gfCNCPoint3[8474] = {X 379.6357, Y 98.2550, Z -3.8333, A 0.000, B 0.000, C 0.000 }
gfCNCPoint3[8475] = {X 377.3857, Y 99.2021, Z -3.8333, A 0.000, B 0.000, C 0.000 }
gfCNCPoint3[8476] = {X 375.0734, Y 99.9850, Z -3.8333, A 0.000, B 0.000, C 0.000 }
gfCNCPoint3[8477] = {X 372.7108, Y 100.5996, Z -3.8333, A 0.000, B 0.000, C 0.000 }
gfCNCPoint3[8478] = {X 368.9146, Y 101.3340, Z -3.8333, A 0.000, B 0.000, C 0.000 }
gfCNCPoint3[8479] = {X 365.0874, Y 101.8851, Z -3.8333, A 0.000, B 0.000, C 0.000 }
gfCNCPoint3[8480] = {X 361.2381, Y 102.2515, Z -3.8333, A 0.000, B 0.000, C 0.000 }
gfCNCPoint3[8481] = {X 357.2381, Y 102.4918, Z -3.8333, A 0.000, B 0.000, C 0.000 }
gfCNCPoint3[8482] = {X 353.2338, Y 102.6450, Z -3.8333, A 0.000, B 0.000, C 0.000 }
gfCNCPoint3[8483] = {X 353.3454, Y 106.7235, Z -3.8333, A 0.000, B 0.000, C 0.000 }
gfCNCPoint3[8484] = {X 353.3454, Y 106.7235, Z -0.8333, A 0.000, B 0.000, C 0.000 }
gfCNCPoint3[8485] = {X 353.3454, Y 106.7235, Z 11.0000, A 0.000, B 0.000, C 0.000 }
gfCNCPoint3[8486] = {X 411.5989, Y 79.5929, Z 11.0000, A 0.000, B 0.000, C 0.000 }
gfCNCPoint3[8487] = {X 411.5989, Y 79.5929, Z -0.8333, A 0.000, B 0.000, C 0.000 }
gfCNCPoint3[8488] = {X 411.5989, Y 79.5929, Z -3.8333, A 0.000, B 0.000, C 0.000 }
gfCNCPoint3[8489] = {X 413.7992, Y 83.0287, Z -3.8333, A 0.000, B 0.000, C 0.000 }
gfCNCPoint3[8490] = {X 428.0548, Y 73.8995, Z -3.8333, A 0.000, B 0.000, C 0.000 }
gfCNCPoint3[8491] = {X 403.7555, Y 64.3655, Z -3.8333, A 0.000, B 0.000, C 0.000 }
gfCNCPoint3[8492] = {X 402.0596, Y 63.8040, Z -3.8333, A 0.000, B 0.000, C 0.000 }
gfCNCPoint3[8493] = {X 400.3124, Y 63.4320, Z -3.8333, A 0.000, B 0.000, C 0.000 }
gfCNCPoint3[8494] = {X 398.5348, Y 63.2540, Z -3.8333, A 0.000, B 0.000, C 0.000 }
gfCNCPoint3[8495] = {X 397.5823, Y 63.1425, Z -3.8333, A 0.000, B 0.000, C 0.000 }
gfCNCPoint3[8496] = {X 396.6778, Y 62.8236, Z -3.8333, A 0.000, B 0.000, C 0.000 }
gfCNCPoint3[8497] = {X 395.8660, Y 62.3130, Z -3.8333, A 0.000, B 0.000, C 0.000 }
gfCNCPoint3[8498] = {X 395.1868, Y 61.6358, Z -3.8333, A 0.000, B 0.000, C 0.000 }
gfCNCPoint3[8499] = {X 394.6738, Y 60.8255, Z -3.8333, A 0.000, B 0.000, C 0.000 }
gfCNCPoint3[8500] = {X 394.3522, Y 59.9220, Z -3.8333, A 0.000, B 0.000, C 0.000 }
gfCNCPoint3[8501] = {X 394.2379, Y 58.9697, Z -3.8333, A 0.000, B 0.000, C 0.000 }
gfCNCPoint3[8502] = {X 394.2377, Y 58.0000, Z -3.8333, A 0.000, B 0.000, C 0.000 }
gfCNCPoint3[8503] = {X 394.3460, Y 57.0387, Z -3.8333, A 0.000, B 0.000, C 0.000 }
gfCNCPoint3[8504] = {X 394.6655, Y 56.1256, Z -3.8333, A 0.000, B 0.000, C 0.000 }
gfCNCPoint3[8505] = {X 395.1802, Y 55.3065, Z -3.8333, A 0.000, B 0.000, C 0.000 }
gfCNCPoint3[8506] = {X 395.8642, Y 54.6225, Z -3.8333, A 0.000, B 0.000, C 0.000 }
gfCNCPoint3[8507] = {X 396.6833, Y 54.1078, Z -3.8333, A 0.000, B 0.000, C 0.000 }
gfCNCPoint3[8508] = {X 397.5964, Y 53.7883, Z -3.8333, A 0.000, B 0.000, C 0.000 }
gfCNCPoint3[8509] = {X 398.5577, Y 53.6800, Z -3.8333, A 0.000, B 0.000, C 0.000 }
gfCNCPoint3[8510] = {X 419.4886, Y 53.6800, Z -3.8333, A 0.000, B 0.000, C 0.000 }
gfCNCPoint3[8511] = {X 420.4499, Y 53.7883, Z -3.8333, A 0.000, B 0.000, C 0.000 }
gfCNCPoint3[8512] = {X 421.3630, Y 54.1078, Z -3.8333, A 0.000, B 0.000, C 0.000 }
gfCNCPoint3[8513] = {X 422.1821, Y 54.6225, Z -3.8333, A 0.000, B 0.000, C 0.000 }
gfCNCPoint3[8514] = {X 422.8661, Y 55.3065, Z -3.8333, A 0.000, B 0.000, C 0.000 }
gfCNCPoint3[8515] = {X 423.3808, Y 56.1256, Z -3.8333, A 0.000, B 0.000, C 0.000 }
gfCNCPoint3[8516] = {X 423.7003, Y 57.0387, Z -3.8333, A 0.000, B 0.000, C 0.000 }
gfCNCPoint3[8517] = {X 423.8086, Y 58.0000, Z -3.8333, A 0.000, B 0.000, C 0.000 }
gfCNCPoint3[8518] = {X 423.8086, Y 58.2323, Z -3.8333, A 0.000, B 0.000, C 0.000 }
gfCNCPoint3[8519] = {X 429.6116, Y 60.4937, Z -3.8333, A 0.000, B 0.000, C 0.000 }
gfCNCPoint3[8520] = {X 457.8588, Y 71.7009, Z -3.8333, A 0.000, B 0.000, C 0.000 }
gfCNCPoint3[8521] = {X 457.8609, Y 63.2124, Z -3.8333, A 0.000, B 0.000, C 0.000 }
gfCNCPoint3[8522] = {X 457.0092, Y 63.0033, Z -3.8333, A 0.000, B 0.000, C 0.000 }
gfCNCPoint3[8523] = {X 456.2172, Y 62.6265, Z -3.8333, A 0.000, B 0.000, C 0.000 }
gfCNCPoint3[8524] = {X 455.5177, Y 62.0976, Z -3.8333, A 0.000, B 0.000, C 0.000 }
gfCNCPoint3[8525] = {X 454.9395, Y 61.4383, Z -3.8333, A 0.000, B 0.000, C 0.000 }
gfCNCPoint3[8526] = {X 454.5063, Y 60.6757, Z -3.8333, A 0.000, B 0.000, C 0.000 }
gfCNCPoint3[8527] = {X 454.2360, Y 59.8414, Z -3.8333, A 0.000, B 0.000, C 0.000 }
gfCNCPoint3[8528] = {X 454.1398, Y 58.9697, Z -3.8333, A 0.000, B 0.000, C 0.000 }
gfCNCPoint3[8529] = {X 454.1396, Y 58.0000, Z -3.8333, A 0.000, B 0.000, C 0.000 }
gfCNCPoint3[8530] = {X 454.2479, Y 57.0387, Z -3.8333, A 0.000, B 0.000, C 0.000 }
gfCNCPoint3[8531] = {X 454.5674, Y 56.1256, Z -3.8333, A 0.000, B 0.000, C 0.000 }
gfCNCPoint3[8532] = {X 455.0821, Y 55.3065, Z -3.8333, A 0.000, B 0.000, C 0.000 }
gfCNCPoint3[8533] = {X 455.7661, Y 54.6225, Z -3.8333, A 0.000, B 0.000, C 0.000 }
gfCNCPoint3[8534] = {X 456.5852, Y 54.1078, Z -3.8333, A 0.000, B 0.000, C 0.000 }
gfCNCPoint3[8535] = {X 457.4983, Y 53.7883, Z -3.8333, A 0.000, B 0.000, C 0.000 }
gfCNCPoint3[8536] = {X 458.4596, Y 53.6800, Z -3.8333, A 0.000, B 0.000, C 0.000 }
gfCNCPoint3[8537] = {X 475.0000, Y 53.6800, Z -3.8333, A 0.000, B 0.000, C 0.000 }
gfCNCPoint3[8538] = {X 475.9613, Y 53.7883, Z -3.8333, A 0.000, B 0.000, C 0.000 }
gfCNCPoint3[8539] = {X 476.8744, Y 54.1078, Z -3.8333, A 0.000, B 0.000, C 0.000 }
gfCNCPoint3[8540] = {X 477.6935, Y 54.6225, Z -3.8333, A 0.000, B 0.000, C 0.000 }
gfCNCPoint3[8541] = {X 478.3775, Y 55.3065, Z -3.8333, A 0.000, B 0.000, C 0.000 }
gfCNCPoint3[8542] = {X 478.8922, Y 56.1256, Z -3.8333, A 0.000, B 0.000, C 0.000 }
gfCNCPoint3[8543] = {X 479.2117, Y 57.0387, Z -3.8333, A 0.000, B 0.000, C 0.000 }
gfCNCPoint3[8544] = {X 479.3200, Y 58.0000, Z -3.8333, A 0.000, B 0.000, C 0.000 }
gfCNCPoint3[8545] = {X 479.3200, Y 58.9342, Z -3.8333, A 0.000, B 0.000, C 0.000 }
gfCNCPoint3[8546] = {X 479.2300, Y 59.8115, Z -3.8333, A 0.000, B 0.000, C 0.000 }
gfCNCPoint3[8547] = {X 478.9637, Y 60.6522, Z -3.8333, A 0.000, B 0.000, C 0.000 }
gfCNCPoint3[8548] = {X 478.5322, Y 61.4212, Z -3.8333, A 0.000, B 0.000, C 0.000 }
gfCNCPoint3[8549] = {X 477.9535, Y 62.0867, Z -3.8333, A 0.000, B 0.000, C 0.000 }
gfCNCPoint3[8550] = {X 477.2518, Y 62.6208, Z -3.8333, A 0.000, B 0.000, C 0.000 }
gfCNCPoint3[8551] = {X 476.4562, Y 63.0012, Z -3.8333, A 0.000, B 0.000, C 0.000 }
gfCNCPoint3[8552] = {X 475.6000, Y 63.2122, Z -3.8333, A 0.000, B 0.000, C 0.000 }
gfCNCPoint3[8553] = {X 475.6004, Y 92.7684, Z -3.8333, A 0.000, B 0.000, C 0.000 }
gfCNCPoint3[8554] = {X 475.9967, Y 92.8675, Z -3.8333, A 0.000, B 0.000, C 0.000 }
gfCNCPoint3[8555] = {X 476.3874, Y 92.9869, Z -3.8333, A 0.000, B 0.000, C 0.000 }
gfCNCPoint3[8556] = {X 477.1991, Y 93.3557, Z -3.8333, A 0.000, B 0.000, C 0.000 }
gfCNCPoint3[8557] = {X 477.9172, Y 93.8843, Z -3.8333, A 0.000, B 0.000, C 0.000 }
gfCNCPoint3[8558] = {X 478.5105, Y 94.5498, Z -3.8333, A 0.000, B 0.000, C 0.000 }
gfCNCPoint3[8559] = {X 478.9537, Y 95.3235, Z -3.8333, A 0.000, B 0.000, C 0.000 }
gfCNCPoint3[8560] = {X 479.2274, Y 96.1721, Z -3.8333, A 0.000, B 0.000, C 0.000 }
gfCNCPoint3[8561] = {X 479.3200, Y 97.0589, Z -3.8333, A 0.000, B 0.000, C 0.000 }
gfCNCPoint3[8562] = {X 479.3200, Y 98.0000, Z -3.8333, A 0.000, B 0.000, C 0.000 }
gfCNCPoint3[8563] = {X 479.2117, Y 98.9613, Z -3.8333, A 0.000, B 0.000, C 0.000 }
gfCNCPoint3[8564] = {X 478.8922, Y 99.8744, Z -3.8333, A 0.000, B 0.000, C 0.000 }
gfCNCPoint3[8565] = {X 478.3775, Y 100.6935, Z -3.8333, A 0.000, B 0.000, C 0.000 }
gfCNCPoint3[8566] = {X 477.6935, Y 101.3775, Z -3.8333, A 0.000, B 0.000, C 0.000 }
gfCNCPoint3[8567] = {X 476.8744, Y 101.8922, Z -3.8333, A 0.000, B 0.000, C 0.000 }
gfCNCPoint3[8568] = {X 475.9613, Y 102.2117, Z -3.8333, A 0.000, B 0.000, C 0.000 }
gfCNCPoint3[8569] = {X 475.0000, Y 102.3200, Z -3.8333, A 0.000, B 0.000, C 0.000 }
gfCNCPoint3[8570] = {X 458.4596, Y 102.3200, Z -3.8333, A 0.000, B 0.000, C 0.000 }
gfCNCPoint3[8571] = {X 457.4983, Y 102.2117, Z -3.8333, A 0.000, B 0.000, C 0.000 }
gfCNCPoint3[8572] = {X 456.5852, Y 101.8922, Z -3.8333, A 0.000, B 0.000, C 0.000 }
gfCNCPoint3[8573] = {X 455.7661, Y 101.3775, Z -3.8333, A 0.000, B 0.000, C 0.000 }
gfCNCPoint3[8574] = {X 455.0821, Y 100.6935, Z -3.8333, A 0.000, B 0.000, C 0.000 }
gfCNCPoint3[8575] = {X 454.5674, Y 99.8744, Z -3.8333, A 0.000, B 0.000, C 0.000 }
gfCNCPoint3[8576] = {X 454.2479, Y 98.9613, Z -3.8333, A 0.000, B 0.000, C 0.000 }
gfCNCPoint3[8577] = {X 454.1396, Y 98.0000, Z -3.8333, A 0.000, B 0.000, C 0.000 }
gfCNCPoint3[8578] = {X 454.1396, Y 97.0659, Z -3.8333, A 0.000, B 0.000, C 0.000 }
gfCNCPoint3[8579] = {X 454.2295, Y 96.1891, Z -3.8333, A 0.000, B 0.000, C 0.000 }
gfCNCPoint3[8580] = {X 454.4955, Y 95.3488, Z -3.8333, A 0.000, B 0.000, C 0.000 }
gfCNCPoint3[8581] = {X 454.9265, Y 94.5800, Z -3.8333, A 0.000, B 0.000, C 0.000 }
gfCNCPoint3[8582] = {X 455.5046, Y 93.9147, Z -3.8333, A 0.000, B 0.000, C 0.000 }
gfCNCPoint3[8583] = {X 456.2057, Y 93.3805, Z -3.8333, A 0.000, B 0.000, C 0.000 }
gfCNCPoint3[8584] = {X 457.0006, Y 92.9998, Z -3.8333, A 0.000, B 0.000, C 0.000 }
gfCNCPoint3[8585] = {X 457.8563, Y 92.7883, Z -3.8333, A 0.000, B 0.000, C 0.000 }
gfCNCPoint3[8586] = {X 457.8563, Y 85.5950, Z -3.8333, A 0.000, B 0.000, C 0.000 }
gfCNCPoint3[8587] = {X 444.8588, Y 80.4999, Z -3.8333, A 0.000, B 0.000, C 0.000 }
gfCNCPoint3[8588] = {X 420.0232, Y 96.5882, Z -3.8333, A 0.000, B 0.000, C 0.000 }
gfCNCPoint3[8589] = {X 420.0267, Y 97.0647, Z -3.8333, A 0.000, B 0.000, C 0.000 }
gfCNCPoint3[8590] = {X 420.0267, Y 98.0000, Z -3.8333, A 0.000, B 0.000, C 0.000 }
gfCNCPoint3[8591] = {X 419.9184, Y 98.9613, Z -3.8333, A 0.000, B 0.000, C 0.000 }
gfCNCPoint3[8592] = {X 419.5989, Y 99.8744, Z -3.8333, A 0.000, B 0.000, C 0.000 }
gfCNCPoint3[8593] = {X 419.0842, Y 100.6935, Z -3.8333, A 0.000, B 0.000, C 0.000 }
gfCNCPoint3[8594] = {X 418.4002, Y 101.3775, Z -3.8333, A 0.000, B 0.000, C 0.000 }
gfCNCPoint3[8595] = {X 417.5811, Y 101.8922, Z -3.8333, A 0.000, B 0.000, C 0.000 }
gfCNCPoint3[8596] = {X 416.6680, Y 102.2117, Z -3.8333, A 0.000, B 0.000, C 0.000 }
gfCNCPoint3[8597] = {X 415.7067, Y 102.3200, Z -3.8333, A 0.000, B 0.000, C 0.000 }
gfCNCPoint3[8598] = {X 396.4059, Y 102.3200, Z -3.8333, A 0.000, B 0.000, C 0.000 }
gfCNCPoint3[8599] = {X 395.4447, Y 102.2117, Z -3.8333, A 0.000, B 0.000, C 0.000 }
gfCNCPoint3[8600] = {X 394.5316, Y 101.8922, Z -3.8333, A 0.000, B 0.000, C 0.000 }
gfCNCPoint3[8601] = {X 393.7125, Y 101.3775, Z -3.8333, A 0.000, B 0.000, C 0.000 }
gfCNCPoint3[8602] = {X 393.0284, Y 100.6935, Z -3.8333, A 0.000, B 0.000, C 0.000 }
gfCNCPoint3[8603] = {X 392.5138, Y 99.8744, Z -3.8333, A 0.000, B 0.000, C 0.000 }
gfCNCPoint3[8604] = {X 392.1943, Y 98.9613, Z -3.8333, A 0.000, B 0.000, C 0.000 }
gfCNCPoint3[8605] = {X 392.0859, Y 98.0000, Z -3.8333, A 0.000, B 0.000, C 0.000 }
gfCNCPoint3[8606] = {X 392.0859, Y 97.0659, Z -3.8333, A 0.000, B 0.000, C 0.000 }
gfCNCPoint3[8607] = {X 392.1954, Y 96.0997, Z -3.8333, A 0.000, B 0.000, C 0.000 }
gfCNCPoint3[8608] = {X 392.5182, Y 95.1825, Z -3.8333, A 0.000, B 0.000, C 0.000 }
gfCNCPoint3[8609] = {X 393.0379, Y 94.3606, Z -3.8333, A 0.000, B 0.000, C 0.000 }
gfCNCPoint3[8610] = {X 393.7283, Y 93.6759, Z -3.8333, A 0.000, B 0.000, C 0.000 }
gfCNCPoint3[8611] = {X 394.5544, Y 93.1629, Z -3.8333, A 0.000, B 0.000, C 0.000 }
gfCNCPoint3[8612] = {X 395.4742, Y 92.8476, Z -3.8333, A 0.000, B 0.000, C 0.000 }
gfCNCPoint3[8613] = {X 396.4413, Y 92.7461, Z -3.8333, A 0.000, B 0.000, C 0.000 }
gfCNCPoint3[8614] = {X 397.3691, Y 92.7028, Z -3.8333, A 0.000, B 0.000, C 0.000 }
gfCNCPoint3[8615] = {X 398.2936, Y 92.6146, Z -3.8333, A 0.000, B 0.000, C 0.000 }
gfCNCPoint3[8616] = {X 398.9444, Y 92.4569, Z -3.8333, A 0.000, B 0.000, C 0.000 }
gfCNCPoint3[8617] = {X 399.5436, Y 92.1580, Z -3.8333, A 0.000, B 0.000, C 0.000 }
gfCNCPoint3[8618] = {X 413.7992, Y 83.0287, Z -3.8333, A 0.000, B 0.000, C 0.000 }
gfCNCPoint3[8619] = {X 411.6421, Y 79.6603, Z -3.8333, A 0.000, B 0.000, C 0.000 }
gfCNCPoint3[8620] = {X 413.8424, Y 83.0961, Z -3.8333, A 0.000, B 0.000, C 0.000 }
gfCNCPoint3[8621] = {X 428.2300, Y 73.8823, Z -3.8333, A 0.000, B 0.000, C 0.000 }
gfCNCPoint3[8622] = {X 403.7847, Y 64.2910, Z -3.8333, A 0.000, B 0.000, C 0.000 }
gfCNCPoint3[8623] = {X 402.0800, Y 63.7266, Z -3.8333, A 0.000, B 0.000, C 0.000 }
gfCNCPoint3[8624] = {X 400.3236, Y 63.3528, Z -3.8333, A 0.000, B 0.000, C 0.000 }
gfCNCPoint3[8625] = {X 398.5368, Y 63.1740, Z -3.8333, A 0.000, B 0.000, C 0.000 }
gfCNCPoint3[8626] = {X 397.6017, Y 63.0649, Z -3.8333, A 0.000, B 0.000, C 0.000 }
gfCNCPoint3[8627] = {X 396.7136, Y 62.7520, Z -3.8333, A 0.000, B 0.000, C 0.000 }
gfCNCPoint3[8628] = {X 395.9165, Y 62.2509, Z -3.8333, A 0.000, B 0.000, C 0.000 }
gfCNCPoint3[8629] = {X 395.2497, Y 61.5863, Z -3.8333, A 0.000, B 0.000, C 0.000 }
gfCNCPoint3[8630] = {X 394.7459, Y 60.7909, Z -3.8333, A 0.000, B 0.000, C 0.000 }
gfCNCPoint3[8631] = {X 394.4301, Y 59.9039, Z -3.8333, A 0.000, B 0.000, C 0.000 }
gfCNCPoint3[8632] = {X 394.3179, Y 58.9691, Z -3.8333, A 0.000, B 0.000, C 0.000 }
gfCNCPoint3[8633] = {X 394.3177, Y 58.0000, Z -3.8333, A 0.000, B 0.000, C 0.000 }
gfCNCPoint3[8634] = {X 394.4240, Y 57.0565, Z -3.8333, A 0.000, B 0.000, C 0.000 }
gfCNCPoint3[8635] = {X 394.7376, Y 56.1603, Z -3.8333, A 0.000, B 0.000, C 0.000 }
gfCNCPoint3[8636] = {X 395.2428, Y 55.3564, Z -3.8333, A 0.000, B 0.000, C 0.000 }
gfCNCPoint3[8637] = {X 395.9141, Y 54.6850, Z -3.8333, A 0.000, B 0.000, C 0.000 }
gfCNCPoint3[8638] = {X 396.7181, Y 54.1799, Z -3.8333, A 0.000, B 0.000, C 0.000 }
gfCNCPoint3[8639] = {X 397.6142, Y 53.8663, Z -3.8333, A 0.000, B 0.000, C 0.000 }
gfCNCPoint3[8640] = {X 398.5577, Y 53.7600, Z -3.8333, A 0.000, B 0.000, C 0.000 }
gfCNCPoint3[8641] = {X 419.4886, Y 53.7600, Z -3.8333, A 0.000, B 0.000, C 0.000 }
gfCNCPoint3[8642] = {X 420.4321, Y 53.8663, Z -3.8333, A 0.000, B 0.000, C 0.000 }
gfCNCPoint3[8643] = {X 421.3283, Y 54.1799, Z -3.8333, A 0.000, B 0.000, C 0.000 }
gfCNCPoint3[8644] = {X 422.1322, Y 54.6850, Z -3.8333, A 0.000, B 0.000, C 0.000 }
gfCNCPoint3[8645] = {X 422.8036, Y 55.3564, Z -3.8333, A 0.000, B 0.000, C 0.000 }
gfCNCPoint3[8646] = {X 423.3087, Y 56.1603, Z -3.8333, A 0.000, B 0.000, C 0.000 }
gfCNCPoint3[8647] = {X 423.6223, Y 57.0565, Z -3.8333, A 0.000, B 0.000, C 0.000 }
gfCNCPoint3[8648] = {X 423.7286, Y 58.0000, Z -3.8333, A 0.000, B 0.000, C 0.000 }
gfCNCPoint3[8649] = {X 423.7286, Y 58.2870, Z -3.8333, A 0.000, B 0.000, C 0.000 }
gfCNCPoint3[8650] = {X 429.5823, Y 60.5682, Z -3.8333, A 0.000, B 0.000, C 0.000 }
gfCNCPoint3[8651] = {X 457.9388, Y 71.8187, Z -3.8333, A 0.000, B 0.000, C 0.000 }
gfCNCPoint3[8652] = {X 457.9409, Y 63.1422, Z -3.8333, A 0.000, B 0.000, C 0.000 }
gfCNCPoint3[8653] = {X 457.0923, Y 62.9476, Z -3.8333, A 0.000, B 0.000, C 0.000 }
gfCNCPoint3[8654] = {X 456.3014, Y 62.5837, Z -3.8333, A 0.000, B 0.000, C 0.000 }
gfCNCPoint3[8655] = {X 455.6014, Y 62.0659, Z -3.8333, A 0.000, B 0.000, C 0.000 }
gfCNCPoint3[8656] = {X 455.0220, Y 61.4161, Z -3.8333, A 0.000, B 0.000, C 0.000 }
gfCNCPoint3[8657] = {X 454.5875, Y 60.6616, Z -3.8333, A 0.000, B 0.000, C 0.000 }
gfCNCPoint3[8658] = {X 454.3163, Y 59.8343, Z -3.8333, A 0.000, B 0.000, C 0.000 }
gfCNCPoint3[8659] = {X 454.2197, Y 58.9691, Z -3.8333, A 0.000, B 0.000, C 0.000 }
gfCNCPoint3[8660] = {X 454.2196, Y 58.0000, Z -3.8333, A 0.000, B 0.000, C 0.000 }
gfCNCPoint3[8661] = {X 454.3259, Y 57.0565, Z -3.8333, A 0.000, B 0.000, C 0.000 }
gfCNCPoint3[8662] = {X 454.6395, Y 56.1603, Z -3.8333, A 0.000, B 0.000, C 0.000 }
gfCNCPoint3[8663] = {X 455.1446, Y 55.3564, Z -3.8333, A 0.000, B 0.000, C 0.000 }
gfCNCPoint3[8664] = {X 455.8160, Y 54.6850, Z -3.8333, A 0.000, B 0.000, C 0.000 }
gfCNCPoint3[8665] = {X 456.6199, Y 54.1799, Z -3.8333, A 0.000, B 0.000, C 0.000 }
gfCNCPoint3[8666] = {X 457.5161, Y 53.8663, Z -3.8333, A 0.000, B 0.000, C 0.000 }
gfCNCPoint3[8667] = {X 458.4596, Y 53.7600, Z -3.8333, A 0.000, B 0.000, C 0.000 }
gfCNCPoint3[8668] = {X 475.0000, Y 53.7600, Z -3.8333, A 0.000, B 0.000, C 0.000 }
gfCNCPoint3[8669] = {X 475.9435, Y 53.8663, Z -3.8333, A 0.000, B 0.000, C 0.000 }
gfCNCPoint3[8670] = {X 476.8397, Y 54.1799, Z -3.8333, A 0.000, B 0.000, C 0.000 }
gfCNCPoint3[8671] = {X 477.6436, Y 54.6850, Z -3.8333, A 0.000, B 0.000, C 0.000 }
gfCNCPoint3[8672] = {X 478.3150, Y 55.3564, Z -3.8333, A 0.000, B 0.000, C 0.000 }
gfCNCPoint3[8673] = {X 478.8201, Y 56.1603, Z -3.8333, A 0.000, B 0.000, C 0.000 }
gfCNCPoint3[8674] = {X 479.1337, Y 57.0565, Z -3.8333, A 0.000, B 0.000, C 0.000 }
gfCNCPoint3[8675] = {X 479.2400, Y 58.0000, Z -3.8333, A 0.000, B 0.000, C 0.000 }
gfCNCPoint3[8676] = {X 479.2400, Y 58.9342, Z -3.8333, A 0.000, B 0.000, C 0.000 }
gfCNCPoint3[8677] = {X 479.1496, Y 59.8049, Z -3.8333, A 0.000, B 0.000, C 0.000 }
gfCNCPoint3[8678] = {X 478.8823, Y 60.6385, Z -3.8333, A 0.000, B 0.000, C 0.000 }
gfCNCPoint3[8679] = {X 478.4495, Y 61.3995, Z -3.8333, A 0.000, B 0.000, C 0.000 }
gfCNCPoint3[8680] = {X 477.8697, Y 62.0553, Z -3.8333, A 0.000, B 0.000, C 0.000 }
gfCNCPoint3[8681] = {X 477.1676, Y 62.5781, Z -3.8333, A 0.000, B 0.000, C 0.000 }
gfCNCPoint3[8682] = {X 476.3730, Y 62.9456, Z -3.8333, A 0.000, B 0.000, C 0.000 }
gfCNCPoint3[8683] = {X 475.5200, Y 63.1421, Z -3.8333, A 0.000, B 0.000, C 0.000 }
gfCNCPoint3[8684] = {X 475.5204, Y 92.8328, Z -3.8333, A 0.000, B 0.000, C 0.000 }
gfCNCPoint3[8685] = {X 475.9444, Y 92.9360, Z -3.8333, A 0.000, B 0.000, C 0.000 }
gfCNCPoint3[8686] = {X 476.3620, Y 93.0628, Z -3.8333, A 0.000, B 0.000, C 0.000 }
gfCNCPoint3[8687] = {X 477.1586, Y 93.4247, Z -3.8333, A 0.000, B 0.000, C 0.000 }
gfCNCPoint3[8688] = {X 477.8633, Y 93.9435, Z -3.8333, A 0.000, B 0.000, C 0.000 }
gfCNCPoint3[8689] = {X 478.4456, Y 94.5966, Z -3.8333, A 0.000, B 0.000, C 0.000 }
gfCNCPoint3[8690] = {X 478.8805, Y 95.3559, Z -3.8333, A 0.000, B 0.000, C 0.000 }
gfCNCPoint3[8691] = {X 479.1491, Y 96.1886, Z -3.8333, A 0.000, B 0.000, C 0.000 }
gfCNCPoint3[8692] = {X 479.2400, Y 97.0589, Z -3.8333, A 0.000, B 0.000, C 0.000 }
gfCNCPoint3[8693] = {X 479.2400, Y 98.0000, Z -3.8333, A 0.000, B 0.000, C 0.000 }
gfCNCPoint3[8694] = {X 479.1337, Y 98.9435, Z -3.8333, A 0.000, B 0.000, C 0.000 }
gfCNCPoint3[8695] = {X 478.8201, Y 99.8397, Z -3.8333, A 0.000, B 0.000, C 0.000 }
gfCNCPoint3[8696] = {X 478.3150, Y 100.6436, Z -3.8333, A 0.000, B 0.000, C 0.000 }
gfCNCPoint3[8697] = {X 477.6436, Y 101.3150, Z -3.8333, A 0.000, B 0.000, C 0.000 }
gfCNCPoint3[8698] = {X 476.8397, Y 101.8201, Z -3.8333, A 0.000, B 0.000, C 0.000 }
gfCNCPoint3[8699] = {X 475.9435, Y 102.1337, Z -3.8333, A 0.000, B 0.000, C 0.000 }
gfCNCPoint3[8700] = {X 475.0000, Y 102.2400, Z -3.8333, A 0.000, B 0.000, C 0.000 }
gfCNCPoint3[8701] = {X 458.4596, Y 102.2400, Z -3.8333, A 0.000, B 0.000, C 0.000 }
gfCNCPoint3[8702] = {X 457.5161, Y 102.1337, Z -3.8333, A 0.000, B 0.000, C 0.000 }
gfCNCPoint3[8703] = {X 456.6199, Y 101.8201, Z -3.8333, A 0.000, B 0.000, C 0.000 }
gfCNCPoint3[8704] = {X 455.8160, Y 101.3150, Z -3.8333, A 0.000, B 0.000, C 0.000 }
gfCNCPoint3[8705] = {X 455.1446, Y 100.6436, Z -3.8333, A 0.000, B 0.000, C 0.000 }
gfCNCPoint3[8706] = {X 454.6395, Y 99.8397, Z -3.8333, A 0.000, B 0.000, C 0.000 }
gfCNCPoint3[8707] = {X 454.3259, Y 98.9435, Z -3.8333, A 0.000, B 0.000, C 0.000 }
gfCNCPoint3[8708] = {X 454.2196, Y 98.0000, Z -3.8333, A 0.000, B 0.000, C 0.000 }
gfCNCPoint3[8709] = {X 454.2196, Y 97.0659, Z -3.8333, A 0.000, B 0.000, C 0.000 }
gfCNCPoint3[8710] = {X 454.3099, Y 96.1957, Z -3.8333, A 0.000, B 0.000, C 0.000 }
gfCNCPoint3[8711] = {X 454.5769, Y 95.3624, Z -3.8333, A 0.000, B 0.000, C 0.000 }
gfCNCPoint3[8712] = {X 455.0092, Y 94.6018, Z -3.8333, A 0.000, B 0.000, C 0.000 }
gfCNCPoint3[8713] = {X 455.5884, Y 93.9460, Z -3.8333, A 0.000, B 0.000, C 0.000 }
gfCNCPoint3[8714] = {X 456.2899, Y 93.4231, Z -3.8333, A 0.000, B 0.000, C 0.000 }
gfCNCPoint3[8715] = {X 457.0838, Y 93.0553, Z -3.8333, A 0.000, B 0.000, C 0.000 }
gfCNCPoint3[8716] = {X 457.9363, Y 92.8584, Z -3.8333, A 0.000, B 0.000, C 0.000 }
gfCNCPoint3[8717] = {X 457.9363, Y 85.5404, Z -3.8333, A 0.000, B 0.000, C 0.000 }
gfCNCPoint3[8718] = {X 444.8498, Y 80.4105, Z -3.8333, A 0.000, B 0.000, C 0.000 }
gfCNCPoint3[8719] = {X 419.9429, Y 96.5449, Z -3.8333, A 0.000, B 0.000, C 0.000 }
gfCNCPoint3[8720] = {X 419.9467, Y 97.0650, Z -3.8333, A 0.000, B 0.000, C 0.000 }
gfCNCPoint3[8721] = {X 419.9467, Y 98.0000, Z -3.8333, A 0.000, B 0.000, C 0.000 }
gfCNCPoint3[8722] = {X 419.8404, Y 98.9435, Z -3.8333, A 0.000, B 0.000, C 0.000 }
gfCNCPoint3[8723] = {X 419.5268, Y 99.8397, Z -3.8333, A 0.000, B 0.000, C 0.000 }
gfCNCPoint3[8724] = {X 419.0217, Y 100.6436, Z -3.8333, A 0.000, B 0.000, C 0.000 }
gfCNCPoint3[8725] = {X 418.3503, Y 101.3150, Z -3.8333, A 0.000, B 0.000, C 0.000 }
gfCNCPoint3[8726] = {X 417.5464, Y 101.8201, Z -3.8333, A 0.000, B 0.000, C 0.000 }
gfCNCPoint3[8727] = {X 416.6502, Y 102.1337, Z -3.8333, A 0.000, B 0.000, C 0.000 }
gfCNCPoint3[8728] = {X 415.7067, Y 102.2400, Z -3.8333, A 0.000, B 0.000, C 0.000 }
gfCNCPoint3[8729] = {X 396.4059, Y 102.2400, Z -3.8333, A 0.000, B 0.000, C 0.000 }
gfCNCPoint3[8730] = {X 395.4625, Y 102.1337, Z -3.8333, A 0.000, B 0.000, C 0.000 }
gfCNCPoint3[8731] = {X 394.5663, Y 101.8201, Z -3.8333, A 0.000, B 0.000, C 0.000 }
gfCNCPoint3[8732] = {X 393.7624, Y 101.3150, Z -3.8333, A 0.000, B 0.000, C 0.000 }
gfCNCPoint3[8733] = {X 393.0910, Y 100.6436, Z -3.8333, A 0.000, B 0.000, C 0.000 }
gfCNCPoint3[8734] = {X 392.5858, Y 99.8397, Z -3.8333, A 0.000, B 0.000, C 0.000 }
gfCNCPoint3[8735] = {X 392.2723, Y 98.9435, Z -3.8333, A 0.000, B 0.000, C 0.000 }
gfCNCPoint3[8736] = {X 392.1659, Y 98.0000, Z -3.8333, A 0.000, B 0.000, C 0.000 }
gfCNCPoint3[8737] = {X 392.1659, Y 97.0659, Z -3.8333, A 0.000, B 0.000, C 0.000 }
gfCNCPoint3[8738] = {X 392.2734, Y 96.1174, Z -3.8333, A 0.000, B 0.000, C 0.000 }
gfCNCPoint3[8739] = {X 392.5903, Y 95.2170, Z -3.8333, A 0.000, B 0.000, C 0.000 }
gfCNCPoint3[8740] = {X 393.1006, Y 94.4103, Z -3.8333, A 0.000, B 0.000, C 0.000 }
gfCNCPoint3[8741] = {X 393.7784, Y 93.7382, Z -3.8333, A 0.000, B 0.000, C 0.000 }
gfCNCPoint3[8742] = {X 394.5894, Y 93.2348, Z -3.8333, A 0.000, B 0.000, C 0.000 }
gfCNCPoint3[8743] = {X 395.4925, Y 92.9255, Z -3.8333, A 0.000, B 0.000, C 0.000 }
gfCNCPoint3[8744] = {X 396.4419, Y 92.8261, Z -3.8333, A 0.000, B 0.000, C 0.000 }
gfCNCPoint3[8745] = {X 397.3742, Y 92.7827, Z -3.8333, A 0.000, B 0.000, C 0.000 }
gfCNCPoint3[8746] = {X 398.3034, Y 92.6940, Z -3.8333, A 0.000, B 0.000, C 0.000 }
gfCNCPoint3[8747] = {X 398.9717, Y 92.5321, Z -3.8333, A 0.000, B 0.000, C 0.000 }
gfCNCPoint3[8748] = {X 399.5871, Y 92.2251, Z -3.8333, A 0.000, B 0.000, C 0.000 }
gfCNCPoint3[8749] = {X 413.8424, Y 83.0961, Z -3.8333, A 0.000, B 0.000, C 0.000 }
gfCNCPoint3[8750] = {X 411.6852, Y 79.7276, Z -3.8333, A 0.000, B 0.000, C 0.000 }
gfCNCPoint3[8751] = {X 413.8855, Y 83.1635, Z -3.8333, A 0.000, B 0.000, C 0.000 }
gfCNCPoint3[8752] = {X 428.4052, Y 73.8651, Z -3.8333, A 0.000, B 0.000, C 0.000 }
gfCNCPoint3[8753] = {X 403.8140, Y 64.2166, Z -3.8333, A 0.000, B 0.000, C 0.000 }
gfCNCPoint3[8754] = {X 402.1004, Y 63.6493, Z -3.8333, A 0.000, B 0.000, C 0.000 }
gfCNCPoint3[8755] = {X 400.3349, Y 63.2736, Z -3.8333, A 0.000, B 0.000, C 0.000 }
gfCNCPoint3[8756] = {X 398.5388, Y 63.0940, Z -3.8333, A 0.000, B 0.000, C 0.000 }
gfCNCPoint3[8757] = {X 397.6210, Y 62.9872, Z -3.8333, A 0.000, B 0.000, C 0.000 }
gfCNCPoint3[8758] = {X 396.7494, Y 62.6805, Z -3.8333, A 0.000, B 0.000, C 0.000 }
gfCNCPoint3[8759] = {X 395.9671, Y 62.1889, Z -3.8333, A 0.000, B 0.000, C 0.000 }
gfCNCPoint3[8760] = {X 395.3125, Y 61.5368, Z -3.8333, A 0.000, B 0.000, C 0.000 }
gfCNCPoint3[8761] = {X 394.8180, Y 60.7562, Z -3.8333, A 0.000, B 0.000, C 0.000 }
gfCNCPoint3[8762] = {X 394.5081, Y 59.8858, Z -3.8333, A 0.000, B 0.000, C 0.000 }
gfCNCPoint3[8763] = {X 394.3979, Y 58.9684, Z -3.8333, A 0.000, B 0.000, C 0.000 }
gfCNCPoint3[8764] = {X 394.3977, Y 58.0000, Z -3.8333, A 0.000, B 0.000, C 0.000 }
gfCNCPoint3[8765] = {X 394.5020, Y 57.0743, Z -3.8333, A 0.000, B 0.000, C 0.000 }
gfCNCPoint3[8766] = {X 394.8097, Y 56.1950, Z -3.8333, A 0.000, B 0.000, C 0.000 }
gfCNCPoint3[8767] = {X 395.3053, Y 55.4063, Z -3.8333, A 0.000, B 0.000, C 0.000 }
gfCNCPoint3[8768] = {X 395.9640, Y 54.7476, Z -3.8333, A 0.000, B 0.000, C 0.000 }
gfCNCPoint3[8769] = {X 396.7528, Y 54.2520, Z -3.8333, A 0.000, B 0.000, C 0.000 }
gfCNCPoint3[8770] = {X 397.6320, Y 53.9443, Z -3.8333, A 0.000, B 0.000, C 0.000 }
gfCNCPoint3[8771] = {X 398.5577, Y 53.8400, Z -3.8333, A 0.000, B 0.000, C 0.000 }
gfCNCPoint3[8772] = {X 419.4886, Y 53.8400, Z -3.8333, A 0.000, B 0.000, C 0.000 }
gfCNCPoint3[8773] = {X 420.4143, Y 53.9443, Z -3.8333, A 0.000, B 0.000, C 0.000 }
gfCNCPoint3[8774] = {X 421.2936, Y 54.2520, Z -3.8333, A 0.000, B 0.000, C 0.000 }
gfCNCPoint3[8775] = {X 422.0823, Y 54.7476, Z -3.8333, A 0.000, B 0.000, C 0.000 }
gfCNCPoint3[8776] = {X 422.7410, Y 55.4063, Z -3.8333, A 0.000, B 0.000, C 0.000 }
gfCNCPoint3[8777] = {X 423.2366, Y 56.1950, Z -3.8333, A 0.000, B 0.000, C 0.000 }
gfCNCPoint3[8778] = {X 423.5443, Y 57.0743, Z -3.8333, A 0.000, B 0.000, C 0.000 }
gfCNCPoint3[8779] = {X 423.6486, Y 58.0000, Z -3.8333, A 0.000, B 0.000, C 0.000 }
gfCNCPoint3[8780] = {X 423.6486, Y 58.3417, Z -3.8333, A 0.000, B 0.000, C 0.000 }
gfCNCPoint3[8781] = {X 429.5531, Y 60.6426, Z -3.8333, A 0.000, B 0.000, C 0.000 }
gfCNCPoint3[8782] = {X 458.0187, Y 71.9365, Z -3.8333, A 0.000, B 0.000, C 0.000 }
gfCNCPoint3[8783] = {X 458.0209, Y 63.0709, Z -3.8333, A 0.000, B 0.000, C 0.000 }
gfCNCPoint3[8784] = {X 457.9185, Y 63.0587, Z -3.8333, A 0.000, B 0.000, C 0.000 }
gfCNCPoint3[8785] = {X 457.8164, Y 63.0440, Z -3.8333, A 0.000, B 0.000, C 0.000 }
gfCNCPoint3[8786] = {X 456.8788, Y 62.7820, Z -3.8333, A 0.000, B 0.000, C 0.000 }
gfCNCPoint3[8787] = {X 456.0278, Y 62.3093, Z -3.8333, A 0.000, B 0.000, C 0.000 }
gfCNCPoint3[8788] = {X 455.3100, Y 61.6517, Z -3.8333, A 0.000, B 0.000, C 0.000 }
gfCNCPoint3[8789] = {X 454.7646, Y 60.8453, Z -3.8333, A 0.000, B 0.000, C 0.000 }
gfCNCPoint3[8790] = {X 454.4216, Y 59.9343, Z -3.8333, A 0.000, B 0.000, C 0.000 }
gfCNCPoint3[8791] = {X 454.2997, Y 58.9684, Z -3.8333, A 0.000, B 0.000, C 0.000 }
gfCNCPoint3[8792] = {X 454.2996, Y 58.0000, Z -3.8333, A 0.000, B 0.000, C 0.000 }
gfCNCPoint3[8793] = {X 454.4039, Y 57.0743, Z -3.8333, A 0.000, B 0.000, C 0.000 }
gfCNCPoint3[8794] = {X 454.7116, Y 56.1950, Z -3.8333, A 0.000, B 0.000, C 0.000 }
gfCNCPoint3[8795] = {X 455.2072, Y 55.4063, Z -3.8333, A 0.000, B 0.000, C 0.000 }
gfCNCPoint3[8796] = {X 455.8659, Y 54.7476, Z -3.8333, A 0.000, B 0.000, C 0.000 }
gfCNCPoint3[8797] = {X 456.6546, Y 54.2520, Z -3.8333, A 0.000, B 0.000, C 0.000 }
gfCNCPoint3[8798] = {X 457.5339, Y 53.9443, Z -3.8333, A 0.000, B 0.000, C 0.000 }
gfCNCPoint3[8799] = {X 458.4596, Y 53.8400, Z -3.8333, A 0.000, B 0.000, C 0.000 }
gfCNCPoint3[8800] = {X 475.0000, Y 53.8400, Z -3.8333, A 0.000, B 0.000, C 0.000 }
gfCNCPoint3[8801] = {X 475.9257, Y 53.9443, Z -3.8333, A 0.000, B 0.000, C 0.000 }
gfCNCPoint3[8802] = {X 476.8050, Y 54.2520, Z -3.8333, A 0.000, B 0.000, C 0.000 }
gfCNCPoint3[8803] = {X 477.5937, Y 54.7476, Z -3.8333, A 0.000, B 0.000, C 0.000 }
gfCNCPoint3[8804] = {X 478.2524, Y 55.4063, Z -3.8333, A 0.000, B 0.000, C 0.000 }
gfCNCPoint3[8805] = {X 478.7480, Y 56.1950, Z -3.8333, A 0.000, B 0.000, C 0.000 }
gfCNCPoint3[8806] = {X 479.0557, Y 57.0743, Z -3.8333, A 0.000, B 0.000, C 0.000 }
gfCNCPoint3[8807] = {X 479.1600, Y 58.0000, Z -3.8333, A 0.000, B 0.000, C 0.000 }
gfCNCPoint3[8808] = {X 479.1600, Y 58.9342, Z -3.8333, A 0.000, B 0.000, C 0.000 }
gfCNCPoint3[8809] = {X 479.0692, Y 59.7984, Z -3.8333, A 0.000, B 0.000, C 0.000 }
gfCNCPoint3[8810] = {X 478.8009, Y 60.6248, Z -3.8333, A 0.000, B 0.000, C 0.000 }
gfCNCPoint3[8811] = {X 478.3668, Y 61.3775, Z -3.8333, A 0.000, B 0.000, C 0.000 }
gfCNCPoint3[8812] = {X 477.7857, Y 62.0236, Z -3.8333, A 0.000, B 0.000, C 0.000 }
gfCNCPoint3[8813] = {X 477.0832, Y 62.5349, Z -3.8333, A 0.000, B 0.000, C 0.000 }
gfCNCPoint3[8814] = {X 476.2897, Y 62.8891, Z -3.8333, A 0.000, B 0.000, C 0.000 }
gfCNCPoint3[8815] = {X 475.4400, Y 63.0707, Z -3.8333, A 0.000, B 0.000, C 0.000 }
gfCNCPoint3[8816] = {X 475.4404, Y 92.8977, Z -3.8333, A 0.000, B 0.000, C 0.000 }
gfCNCPoint3[8817] = {X 475.8921, Y 93.0047, Z -3.8333, A 0.000, B 0.000, C 0.000 }
gfCNCPoint3[8818] = {X 476.3367, Y 93.1386, Z -3.8333, A 0.000, B 0.000, C 0.000 }
gfCNCPoint3[8819] = {X 477.1182, Y 93.4938, Z -3.8333, A 0.000, B 0.000, C 0.000 }
gfCNCPoint3[8820] = {X 477.8094, Y 94.0026, Z -3.8333, A 0.000, B 0.000, C 0.000 }
gfCNCPoint3[8821] = {X 478.3807, Y 94.6433, Z -3.8333, A 0.000, B 0.000, C 0.000 }
gfCNCPoint3[8822] = {X 478.8073, Y 95.3882, Z -3.8333, A 0.000, B 0.000, C 0.000 }
gfCNCPoint3[8823] = {X 479.0709, Y 96.2051, Z -3.8333, A 0.000, B 0.000, C 0.000 }
gfCNCPoint3[8824] = {X 479.1600, Y 97.0589, Z -3.8333, A 0.000, B 0.000, C 0.000 }
gfCNCPoint3[8825] = {X 479.1600, Y 98.0000, Z -3.8333, A 0.000, B 0.000, C 0.000 }
gfCNCPoint3[8826] = {X 479.0557, Y 98.9257, Z -3.8333, A 0.000, B 0.000, C 0.000 }
gfCNCPoint3[8827] = {X 478.7480, Y 99.8050, Z -3.8333, A 0.000, B 0.000, C 0.000 }
gfCNCPoint3[8828] = {X 478.2524, Y 100.5937, Z -3.8333, A 0.000, B 0.000, C 0.000 }
gfCNCPoint3[8829] = {X 477.5937, Y 101.2524, Z -3.8333, A 0.000, B 0.000, C 0.000 }
gfCNCPoint3[8830] = {X 476.8050, Y 101.7480, Z -3.8333, A 0.000, B 0.000, C 0.000 }
gfCNCPoint3[8831] = {X 475.9257, Y 102.0557, Z -3.8333, A 0.000, B 0.000, C 0.000 }
gfCNCPoint3[8832] = {X 475.0000, Y 102.1600, Z -3.8333, A 0.000, B 0.000, C 0.000 }
gfCNCPoint3[8833] = {X 458.4596, Y 102.1600, Z -3.8333, A 0.000, B 0.000, C 0.000 }
gfCNCPoint3[8834] = {X 457.5339, Y 102.0557, Z -3.8333, A 0.000, B 0.000, C 0.000 }
gfCNCPoint3[8835] = {X 456.6546, Y 101.7480, Z -3.8333, A 0.000, B 0.000, C 0.000 }
gfCNCPoint3[8836] = {X 455.8659, Y 101.2524, Z -3.8333, A 0.000, B 0.000, C 0.000 }
gfCNCPoint3[8837] = {X 455.2072, Y 100.5937, Z -3.8333, A 0.000, B 0.000, C 0.000 }
gfCNCPoint3[8838] = {X 454.7116, Y 99.8050, Z -3.8333, A 0.000, B 0.000, C 0.000 }
gfCNCPoint3[8839] = {X 454.4039, Y 98.9257, Z -3.8333, A 0.000, B 0.000, C 0.000 }
gfCNCPoint3[8840] = {X 454.2996, Y 98.0000, Z -3.8333, A 0.000, B 0.000, C 0.000 }
gfCNCPoint3[8841] = {X 454.2996, Y 97.0659, Z -3.8333, A 0.000, B 0.000, C 0.000 }
gfCNCPoint3[8842] = {X 454.3903, Y 96.2022, Z -3.8333, A 0.000, B 0.000, C 0.000 }
gfCNCPoint3[8843] = {X 454.6583, Y 95.3761, Z -3.8333, A 0.000, B 0.000, C 0.000 }
gfCNCPoint3[8844] = {X 455.0920, Y 94.6237, Z -3.8333, A 0.000, B 0.000, C 0.000 }
gfCNCPoint3[8845] = {X 455.6724, Y 93.9777, Z -3.8333, A 0.000, B 0.000, C 0.000 }
gfCNCPoint3[8846] = {X 456.3743, Y 93.4663, Z -3.8333, A 0.000, B 0.000, C 0.000 }
gfCNCPoint3[8847] = {X 457.1672, Y 93.1118, Z -3.8333, A 0.000, B 0.000, C 0.000 }
gfCNCPoint3[8848] = {X 458.0163, Y 92.9296, Z -3.8333, A 0.000, B 0.000, C 0.000 }
gfCNCPoint3[8849] = {X 458.0163, Y 85.4858, Z -3.8333, A 0.000, B 0.000, C 0.000 }
gfCNCPoint3[8850] = {X 444.8407, Y 80.3210, Z -3.8333, A 0.000, B 0.000, C 0.000 }
gfCNCPoint3[8851] = {X 419.8626, Y 96.5016, Z -3.8333, A 0.000, B 0.000, C 0.000 }
gfCNCPoint3[8852] = {X 419.8667, Y 97.0653, Z -3.8333, A 0.000, B 0.000, C 0.000 }
gfCNCPoint3[8853] = {X 419.8667, Y 98.0000, Z -3.8333, A 0.000, B 0.000, C 0.000 }
gfCNCPoint3[8854] = {X 419.7624, Y 98.9257, Z -3.8333, A 0.000, B 0.000, C 0.000 }
gfCNCPoint3[8855] = {X 419.4547, Y 99.8050, Z -3.8333, A 0.000, B 0.000, C 0.000 }
gfCNCPoint3[8856] = {X 418.9591, Y 100.5937, Z -3.8333, A 0.000, B 0.000, C 0.000 }
gfCNCPoint3[8857] = {X 418.3004, Y 101.2524, Z -3.8333, A 0.000, B 0.000, C 0.000 }
gfCNCPoint3[8858] = {X 417.5117, Y 101.7480, Z -3.8333, A 0.000, B 0.000, C 0.000 }
gfCNCPoint3[8859] = {X 416.6324, Y 102.0557, Z -3.8333, A 0.000, B 0.000, C 0.000 }
gfCNCPoint3[8860] = {X 415.7067, Y 102.1600, Z -3.8333, A 0.000, B 0.000, C 0.000 }
gfCNCPoint3[8861] = {X 396.4059, Y 102.1600, Z -3.8333, A 0.000, B 0.000, C 0.000 }
gfCNCPoint3[8862] = {X 395.4803, Y 102.0557, Z -3.8333, A 0.000, B 0.000, C 0.000 }
gfCNCPoint3[8863] = {X 394.6010, Y 101.7480, Z -3.8333, A 0.000, B 0.000, C 0.000 }
gfCNCPoint3[8864] = {X 393.8122, Y 101.2524, Z -3.8333, A 0.000, B 0.000, C 0.000 }
gfCNCPoint3[8865] = {X 393.1535, Y 100.5937, Z -3.8333, A 0.000, B 0.000, C 0.000 }
gfCNCPoint3[8866] = {X 392.6579, Y 99.8050, Z -3.8333, A 0.000, B 0.000, C 0.000 }
gfCNCPoint3[8867] = {X 392.3502, Y 98.9257, Z -3.8333, A 0.000, B 0.000, C 0.000 }
gfCNCPoint3[8868] = {X 392.2459, Y 98.0000, Z -3.8333, A 0.000, B 0.000, C 0.000 }
gfCNCPoint3[8869] = {X 392.2459, Y 97.0659, Z -3.8333, A 0.000, B 0.000, C 0.000 }
gfCNCPoint3[8870] = {X 392.3514, Y 96.1352, Z -3.8333, A 0.000, B 0.000, C 0.000 }
gfCNCPoint3[8871] = {X 392.6625, Y 95.2516, Z -3.8333, A 0.000, B 0.000, C 0.000 }
gfCNCPoint3[8872] = {X 393.1633, Y 94.4600, Z -3.8333, A 0.000, B 0.000, C 0.000 }
gfCNCPoint3[8873] = {X 393.8286, Y 93.8006, Z -3.8333, A 0.000, B 0.000, C 0.000 }
gfCNCPoint3[8874] = {X 394.6245, Y 93.3067, Z -3.8333, A 0.000, B 0.000, C 0.000 }
gfCNCPoint3[8875] = {X 395.5108, Y 93.0034, Z -3.8333, A 0.000, B 0.000, C 0.000 }
gfCNCPoint3[8876] = {X 396.4424, Y 92.9061, Z -3.8333, A 0.000, B 0.000, C 0.000 }
gfCNCPoint3[8877] = {X 397.3794, Y 92.8625, Z -3.8333, A 0.000, B 0.000, C 0.000 }
gfCNCPoint3[8878] = {X 398.3132, Y 92.7734, Z -3.8333, A 0.000, B 0.000, C 0.000 }
gfCNCPoint3[8879] = {X 398.9991, Y 92.6073, Z -3.8333, A 0.000, B 0.000, C 0.000 }
gfCNCPoint3[8880] = {X 399.6306, Y 92.2923, Z -3.8333, A 0.000, B 0.000, C 0.000 }
gfCNCPoint3[8881] = {X 413.8855, Y 83.1635, Z -3.8333, A 0.000, B 0.000, C 0.000 }
gfCNCPoint3[8882] = {X 411.7283, Y 79.7950, Z -3.8333, A 0.000, B 0.000, C 0.000 }
gfCNCPoint3[8883] = {X 413.9286, Y 83.2309, Z -3.8333, A 0.000, B 0.000, C 0.000 }
gfCNCPoint3[8884] = {X 428.5804, Y 73.8479, Z -3.8333, A 0.000, B 0.000, C 0.000 }
gfCNCPoint3[8885] = {X 403.8433, Y 64.1422, Z -3.8333, A 0.000, B 0.000, C 0.000 }
gfCNCPoint3[8886] = {X 402.1209, Y 63.5719, Z -3.8333, A 0.000, B 0.000, C 0.000 }
gfCNCPoint3[8887] = {X 400.3462, Y 63.1944, Z -3.8333, A 0.000, B 0.000, C 0.000 }
gfCNCPoint3[8888] = {X 398.5408, Y 63.0140, Z -3.8333, A 0.000, B 0.000, C 0.000 }
gfCNCPoint3[8889] = {X 397.6404, Y 62.9096, Z -3.8333, A 0.000, B 0.000, C 0.000 }
gfCNCPoint3[8890] = {X 396.7852, Y 62.6089, Z -3.8333, A 0.000, B 0.000, C 0.000 }
gfCNCPoint3[8891] = {X 396.0176, Y 62.1269, Z -3.8333, A 0.000, B 0.000, C 0.000 }
gfCNCPoint3[8892] = {X 395.3753, Y 61.4873, Z -3.8333, A 0.000, B 0.000, C 0.000 }
gfCNCPoint3[8893] = {X 394.8902, Y 60.7216, Z -3.8333, A 0.000, B 0.000, C 0.000 }
gfCNCPoint3[8894] = {X 394.5860, Y 59.8677, Z -3.8333, A 0.000, B 0.000, C 0.000 }
gfCNCPoint3[8895] = {X 394.4779, Y 58.9678, Z -3.8333, A 0.000, B 0.000, C 0.000 }
gfCNCPoint3[8896] = {X 394.4777, Y 58.0000, Z -3.8333, A 0.000, B 0.000, C 0.000 }
gfCNCPoint3[8897] = {X 394.5800, Y 57.0921, Z -3.8333, A 0.000, B 0.000, C 0.000 }
gfCNCPoint3[8898] = {X 394.8818, Y 56.2298, Z -3.8333, A 0.000, B 0.000, C 0.000 }
gfCNCPoint3[8899] = {X 395.3679, Y 55.4562, Z -3.8333, A 0.000, B 0.000, C 0.000 }
gfCNCPoint3[8900] = {X 396.0139, Y 54.8101, Z -3.8333, A 0.000, B 0.000, C 0.000 }
gfCNCPoint3[8901] = {X 396.7875, Y 54.3240, Z -3.8333, A 0.000, B 0.000, C 0.000 }
gfCNCPoint3[8902] = {X 397.6498, Y 54.0223, Z -3.8333, A 0.000, B 0.000, C 0.000 }
gfCNCPoint3[8903] = {X 398.5577, Y 53.9200, Z -3.8333, A 0.000, B 0.000, C 0.000 }
gfCNCPoint3[8904] = {X 419.4886, Y 53.9200, Z -3.8333, A 0.000, B 0.000, C 0.000 }
gfCNCPoint3[8905] = {X 420.3965, Y 54.0223, Z -3.8333, A 0.000, B 0.000, C 0.000 }
gfCNCPoint3[8906] = {X 421.2588, Y 54.3240, Z -3.8333, A 0.000, B 0.000, C 0.000 }
gfCNCPoint3[8907] = {X 422.0324, Y 54.8101, Z -3.8333, A 0.000, B 0.000, C 0.000 }
gfCNCPoint3[8908] = {X 422.6785, Y 55.4562, Z -3.8333, A 0.000, B 0.000, C 0.000 }
gfCNCPoint3[8909] = {X 423.1646, Y 56.2298, Z -3.8333, A 0.000, B 0.000, C 0.000 }
gfCNCPoint3[8910] = {X 423.4663, Y 57.0921, Z -3.8333, A 0.000, B 0.000, C 0.000 }
gfCNCPoint3[8911] = {X 423.5686, Y 58.0000, Z -3.8333, A 0.000, B 0.000, C 0.000 }
gfCNCPoint3[8912] = {X 423.5686, Y 58.3964, Z -3.8333, A 0.000, B 0.000, C 0.000 }
gfCNCPoint3[8913] = {X 429.5238, Y 60.7171, Z -3.8333, A 0.000, B 0.000, C 0.000 }
gfCNCPoint3[8914] = {X 458.0987, Y 72.0543, Z -3.8333, A 0.000, B 0.000, C 0.000 }
gfCNCPoint3[8915] = {X 458.1009, Y 62.9983, Z -3.8333, A 0.000, B 0.000, C 0.000 }
gfCNCPoint3[8916] = {X 457.9646, Y 62.9839, Z -3.8333, A 0.000, B 0.000, C 0.000 }
gfCNCPoint3[8917] = {X 457.8288, Y 62.9650, Z -3.8333, A 0.000, B 0.000, C 0.000 }
gfCNCPoint3[8918] = {X 456.9092, Y 62.7080, Z -3.8333, A 0.000, B 0.000, C 0.000 }
gfCNCPoint3[8919] = {X 456.0746, Y 62.2444, Z -3.8333, A 0.000, B 0.000, C 0.000 }
gfCNCPoint3[8920] = {X 455.3706, Y 61.5994, Z -3.8333, A 0.000, B 0.000, C 0.000 }
gfCNCPoint3[8921] = {X 454.8357, Y 60.8086, Z -3.8333, A 0.000, B 0.000, C 0.000 }
gfCNCPoint3[8922] = {X 454.4993, Y 59.9150, Z -3.8333, A 0.000, B 0.000, C 0.000 }
gfCNCPoint3[8923] = {X 454.3797, Y 58.9678, Z -3.8333, A 0.000, B 0.000, C 0.000 }
gfCNCPoint3[8924] = {X 454.3796, Y 58.0000, Z -3.8333, A 0.000, B 0.000, C 0.000 }
gfCNCPoint3[8925] = {X 454.4819, Y 57.0921, Z -3.8333, A 0.000, B 0.000, C 0.000 }
gfCNCPoint3[8926] = {X 454.7837, Y 56.2298, Z -3.8333, A 0.000, B 0.000, C 0.000 }
gfCNCPoint3[8927] = {X 455.2697, Y 55.4562, Z -3.8333, A 0.000, B 0.000, C 0.000 }
gfCNCPoint3[8928] = {X 455.9158, Y 54.8101, Z -3.8333, A 0.000, B 0.000, C 0.000 }
gfCNCPoint3[8929] = {X 456.6894, Y 54.3240, Z -3.8333, A 0.000, B 0.000, C 0.000 }
gfCNCPoint3[8930] = {X 457.5517, Y 54.0223, Z -3.8333, A 0.000, B 0.000, C 0.000 }
gfCNCPoint3[8931] = {X 458.4596, Y 53.9200, Z -3.8333, A 0.000, B 0.000, C 0.000 }
gfCNCPoint3[8932] = {X 475.0000, Y 53.9200, Z -3.8333, A 0.000, B 0.000, C 0.000 }
gfCNCPoint3[8933] = {X 475.9079, Y 54.0223, Z -3.8333, A 0.000, B 0.000, C 0.000 }
gfCNCPoint3[8934] = {X 476.7702, Y 54.3240, Z -3.8333, A 0.000, B 0.000, C 0.000 }
gfCNCPoint3[8935] = {X 477.5438, Y 54.8101, Z -3.8333, A 0.000, B 0.000, C 0.000 }
gfCNCPoint3[8936] = {X 478.1899, Y 55.4562, Z -3.8333, A 0.000, B 0.000, C 0.000 }
gfCNCPoint3[8937] = {X 478.6760, Y 56.2298, Z -3.8333, A 0.000, B 0.000, C 0.000 }
gfCNCPoint3[8938] = {X 478.9777, Y 57.0921, Z -3.8333, A 0.000, B 0.000, C 0.000 }
gfCNCPoint3[8939] = {X 479.0800, Y 58.0000, Z -3.8333, A 0.000, B 0.000, C 0.000 }
gfCNCPoint3[8940] = {X 479.0800, Y 58.9342, Z -3.8333, A 0.000, B 0.000, C 0.000 }
gfCNCPoint3[8941] = {X 478.9888, Y 59.7918, Z -3.8333, A 0.000, B 0.000, C 0.000 }
gfCNCPoint3[8942] = {X 478.7194, Y 60.6111, Z -3.8333, A 0.000, B 0.000, C 0.000 }
gfCNCPoint3[8943] = {X 478.2838, Y 61.3554, Z -3.8333, A 0.000, B 0.000, C 0.000 }
gfCNCPoint3[8944] = {X 477.7015, Y 61.9916, Z -3.8333, A 0.000, B 0.000, C 0.000 }
gfCNCPoint3[8945] = {X 476.9985, Y 62.4911, Z -3.8333, A 0.000, B 0.000, C 0.000 }
gfCNCPoint3[8946] = {X 476.2062, Y 62.8317, Z -3.8333, A 0.000, B 0.000, C 0.000 }
gfCNCPoint3[8947] = {X 475.3600, Y 62.9982, Z -3.8333, A 0.000, B 0.000, C 0.000 }
gfCNCPoint3[8948] = {X 475.3604, Y 92.9632, Z -3.8333, A 0.000, B 0.000, C 0.000 }
gfCNCPoint3[8949] = {X 475.8399, Y 93.0736, Z -3.8333, A 0.000, B 0.000, C 0.000 }
gfCNCPoint3[8950] = {X 476.3113, Y 93.2145, Z -3.8333, A 0.000, B 0.000, C 0.000 }
gfCNCPoint3[8951] = {X 477.0777, Y 93.5628, Z -3.8333, A 0.000, B 0.000, C 0.000 }
gfCNCPoint3[8952] = {X 477.7556, Y 94.0618, Z -3.8333, A 0.000, B 0.000, C 0.000 }
gfCNCPoint3[8953] = {X 478.3158, Y 94.6901, Z -3.8333, A 0.000, B 0.000, C 0.000 }
gfCNCPoint3[8954] = {X 478.7341, Y 95.4205, Z -3.8333, A 0.000, B 0.000, C 0.000 }
gfCNCPoint3[8955] = {X 478.9926, Y 96.2216, Z -3.8333, A 0.000, B 0.000, C 0.000 }
gfCNCPoint3[8956] = {X 479.0800, Y 97.0589, Z -3.8333, A 0.000, B 0.000, C 0.000 }
gfCNCPoint3[8957] = {X 479.0800, Y 98.0000, Z -3.8333, A 0.000, B 0.000, C 0.000 }
gfCNCPoint3[8958] = {X 478.9777, Y 98.9079, Z -3.8333, A 0.000, B 0.000, C 0.000 }
gfCNCPoint3[8959] = {X 478.6760, Y 99.7702, Z -3.8333, A 0.000, B 0.000, C 0.000 }
gfCNCPoint3[8960] = {X 478.1899, Y 100.5438, Z -3.8333, A 0.000, B 0.000, C 0.000 }
gfCNCPoint3[8961] = {X 477.5438, Y 101.1899, Z -3.8333, A 0.000, B 0.000, C 0.000 }
gfCNCPoint3[8962] = {X 476.7702, Y 101.6760, Z -3.8333, A 0.000, B 0.000, C 0.000 }
gfCNCPoint3[8963] = {X 475.9079, Y 101.9777, Z -3.8333, A 0.000, B 0.000, C 0.000 }
gfCNCPoint3[8964] = {X 475.0000, Y 102.0800, Z -3.8333, A 0.000, B 0.000, C 0.000 }
gfCNCPoint3[8965] = {X 458.4596, Y 102.0800, Z -3.8333, A 0.000, B 0.000, C 0.000 }
gfCNCPoint3[8966] = {X 457.5517, Y 101.9777, Z -3.8333, A 0.000, B 0.000, C 0.000 }
gfCNCPoint3[8967] = {X 456.6894, Y 101.6760, Z -3.8333, A 0.000, B 0.000, C 0.000 }
gfCNCPoint3[8968] = {X 455.9158, Y 101.1899, Z -3.8333, A 0.000, B 0.000, C 0.000 }
gfCNCPoint3[8969] = {X 455.2697, Y 100.5438, Z -3.8333, A 0.000, B 0.000, C 0.000 }
gfCNCPoint3[8970] = {X 454.7837, Y 99.7702, Z -3.8333, A 0.000, B 0.000, C 0.000 }
gfCNCPoint3[8971] = {X 454.4819, Y 98.9079, Z -3.8333, A 0.000, B 0.000, C 0.000 }
gfCNCPoint3[8972] = {X 454.3796, Y 98.0000, Z -3.8333, A 0.000, B 0.000, C 0.000 }
gfCNCPoint3[8973] = {X 454.3796, Y 97.0659, Z -3.8333, A 0.000, B 0.000, C 0.000 }
gfCNCPoint3[8974] = {X 454.4707, Y 96.2088, Z -3.8333, A 0.000, B 0.000, C 0.000 }
gfCNCPoint3[8975] = {X 454.7398, Y 95.3899, Z -3.8333, A 0.000, B 0.000, C 0.000 }
gfCNCPoint3[8976] = {X 455.1749, Y 94.6458, Z -3.8333, A 0.000, B 0.000, C 0.000 }
gfCNCPoint3[8977] = {X 455.7566, Y 94.0098, Z -3.8333, A 0.000, B 0.000, C 0.000 }
gfCNCPoint3[8978] = {X 456.4590, Y 93.5101, Z -3.8333, A 0.000, B 0.000, C 0.000 }
gfCNCPoint3[8979] = {X 457.2507, Y 93.1692, Z -3.8333, A 0.000, B 0.000, C 0.000 }
gfCNCPoint3[8980] = {X 458.0963, Y 93.0021, Z -3.8333, A 0.000, B 0.000, C 0.000 }
gfCNCPoint3[8981] = {X 458.0963, Y 85.4313, Z -3.8333, A 0.000, B 0.000, C 0.000 }
gfCNCPoint3[8982] = {X 444.8317, Y 80.2315, Z -3.8333, A 0.000, B 0.000, C 0.000 }
gfCNCPoint3[8983] = {X 419.7823, Y 96.4583, Z -3.8333, A 0.000, B 0.000, C 0.000 }
gfCNCPoint3[8984] = {X 419.7867, Y 97.0656, Z -3.8333, A 0.000, B 0.000, C 0.000 }
gfCNCPoint3[8985] = {X 419.7867, Y 98.0000, Z -3.8333, A 0.000, B 0.000, C 0.000 }
gfCNCPoint3[8986] = {X 419.6844, Y 98.9079, Z -3.8333, A 0.000, B 0.000, C 0.000 }
gfCNCPoint3[8987] = {X 419.3827, Y 99.7702, Z -3.8333, A 0.000, B 0.000, C 0.000 }
gfCNCPoint3[8988] = {X 418.8966, Y 100.5438, Z -3.8333, A 0.000, B 0.000, C 0.000 }
gfCNCPoint3[8989] = {X 418.2505, Y 101.1899, Z -3.8333, A 0.000, B 0.000, C 0.000 }
gfCNCPoint3[8990] = {X 417.4769, Y 101.6760, Z -3.8333, A 0.000, B 0.000, C 0.000 }
gfCNCPoint3[8991] = {X 416.6146, Y 101.9777, Z -3.8333, A 0.000, B 0.000, C 0.000 }
gfCNCPoint3[8992] = {X 415.7067, Y 102.0800, Z -3.8333, A 0.000, B 0.000, C 0.000 }
gfCNCPoint3[8993] = {X 396.4059, Y 102.0800, Z -3.8333, A 0.000, B 0.000, C 0.000 }
gfCNCPoint3[8994] = {X 395.4981, Y 101.9777, Z -3.8333, A 0.000, B 0.000, C 0.000 }
gfCNCPoint3[8995] = {X 394.6357, Y 101.6760, Z -3.8333, A 0.000, B 0.000, C 0.000 }
gfCNCPoint3[8996] = {X 393.8621, Y 101.1899, Z -3.8333, A 0.000, B 0.000, C 0.000 }
gfCNCPoint3[8997] = {X 393.2161, Y 100.5438, Z -3.8333, A 0.000, B 0.000, C 0.000 }
gfCNCPoint3[8998] = {X 392.7300, Y 99.7702, Z -3.8333, A 0.000, B 0.000, C 0.000 }
gfCNCPoint3[8999] = {X 392.4282, Y 98.9079, Z -3.8333, A 0.000, B 0.000, C 0.000 }
gfCNCPoint3[9000] = {X 392.3259, Y 98.0000, Z -3.8333, A 0.000, B 0.000, C 0.000 }
gfCNCPoint3[9001] = {X 392.3259, Y 97.0659, Z -3.8333, A 0.000, B 0.000, C 0.000 }
gfCNCPoint3[9002] = {X 392.4294, Y 96.1529, Z -3.8333, A 0.000, B 0.000, C 0.000 }
gfCNCPoint3[9003] = {X 392.7346, Y 95.2862, Z -3.8333, A 0.000, B 0.000, C 0.000 }
gfCNCPoint3[9004] = {X 393.2260, Y 94.5097, Z -3.8333, A 0.000, B 0.000, C 0.000 }
gfCNCPoint3[9005] = {X 393.8787, Y 93.8629, Z -3.8333, A 0.000, B 0.000, C 0.000 }
gfCNCPoint3[9006] = {X 394.6596, Y 93.3786, Z -3.8333, A 0.000, B 0.000, C 0.000 }
gfCNCPoint3[9007] = {X 395.5290, Y 93.0813, Z -3.8333, A 0.000, B 0.000, C 0.000 }
gfCNCPoint3[9008] = {X 396.4430, Y 92.9861, Z -3.8333, A 0.000, B 0.000, C 0.000 }
gfCNCPoint3[9009] = {X 397.3846, Y 92.9423, Z -3.8333, A 0.000, B 0.000, C 0.000 }
gfCNCPoint3[9010] = {X 398.3230, Y 92.8528, Z -3.8333, A 0.000, B 0.000, C 0.000 }
gfCNCPoint3[9011] = {X 399.0265, Y 92.6825, Z -3.8333, A 0.000, B 0.000, C 0.000 }
gfCNCPoint3[9012] = {X 399.6742, Y 92.3594, Z -3.8333, A 0.000, B 0.000, C 0.000 }
gfCNCPoint3[9013] = {X 413.9286, Y 83.2309, Z -3.8333, A 0.000, B 0.000, C 0.000 }
gfCNCPoint3[9014] = {X 411.7650, Y 79.8523, Z -3.8333, A 0.000, B 0.000, C 0.000 }
gfCNCPoint3[9015] = {X 411.7673, Y 79.8508, Z -3.8333, A 0.000, B 0.000, C 0.000 }
gfCNCPoint3[9016] = {X 413.9653, Y 83.2882, Z -3.8333, A 0.000, B 0.000, C 0.000 }
gfCNCPoint3[9017] = {X 428.7557, Y 73.8307, Z -3.8333, A 0.000, B 0.000, C 0.000 }
gfCNCPoint3[9018] = {X 403.8726, Y 64.0677, Z -3.8333, A 0.000, B 0.000, C 0.000 }
gfCNCPoint3[9019] = {X 402.1413, Y 63.4946, Z -3.8333, A 0.000, B 0.000, C 0.000 }
gfCNCPoint3[9020] = {X 400.3574, Y 63.1151, Z -3.8333, A 0.000, B 0.000, C 0.000 }
gfCNCPoint3[9021] = {X 398.5427, Y 62.9340, Z -3.8333, A 0.000, B 0.000, C 0.000 }
gfCNCPoint3[9022] = {X 397.6551, Y 62.8309, Z -3.8333, A 0.000, B 0.000, C 0.000 }
gfCNCPoint3[9023] = {X 396.8125, Y 62.5333, Z -3.8333, A 0.000, B 0.000, C 0.000 }
gfCNCPoint3[9024] = {X 396.0571, Y 62.0560, Z -3.8333, A 0.000, B 0.000, C 0.000 }
gfCNCPoint3[9025] = {X 395.4264, Y 61.4230, Z -3.8333, A 0.000, B 0.000, C 0.000 }
gfCNCPoint3[9026] = {X 394.9520, Y 60.6657, Z -3.8333, A 0.000, B 0.000, C 0.000 }
gfCNCPoint3[9027] = {X 394.6575, Y 59.8220, Z -3.8333, A 0.000, B 0.000, C 0.000 }
gfCNCPoint3[9028] = {X 394.5577, Y 58.9340, Z -3.8333, A 0.000, B 0.000, C 0.000 }
gfCNCPoint3[9029] = {X 394.5577, Y 58.0000, Z -3.8333, A 0.000, B 0.000, C 0.000 }
gfCNCPoint3[9030] = {X 394.6580, Y 57.1099, Z -3.8333, A 0.000, B 0.000, C 0.000 }
gfCNCPoint3[9031] = {X 394.9538, Y 56.2645, Z -3.8333, A 0.000, B 0.000, C 0.000 }
gfCNCPoint3[9032] = {X 395.4304, Y 55.5060, Z -3.8333, A 0.000, B 0.000, C 0.000 }
gfCNCPoint3[9033] = {X 396.0638, Y 54.8727, Z -3.8333, A 0.000, B 0.000, C 0.000 }
gfCNCPoint3[9034] = {X 396.8222, Y 54.3961, Z -3.8333, A 0.000, B 0.000, C 0.000 }
gfCNCPoint3[9035] = {X 397.6676, Y 54.1003, Z -3.8333, A 0.000, B 0.000, C 0.000 }
gfCNCPoint3[9036] = {X 398.5577, Y 54.0000, Z -3.8333, A 0.000, B 0.000, C 0.000 }
gfCNCPoint3[9037] = {X 419.4886, Y 54.0000, Z -3.8333, A 0.000, B 0.000, C 0.000 }
gfCNCPoint3[9038] = {X 420.3787, Y 54.1003, Z -3.8333, A 0.000, B 0.000, C 0.000 }
gfCNCPoint3[9039] = {X 421.2241, Y 54.3961, Z -3.8333, A 0.000, B 0.000, C 0.000 }
gfCNCPoint3[9040] = {X 421.9826, Y 54.8727, Z -3.8333, A 0.000, B 0.000, C 0.000 }
gfCNCPoint3[9041] = {X 422.6159, Y 55.5060, Z -3.8333, A 0.000, B 0.000, C 0.000 }
gfCNCPoint3[9042] = {X 423.0925, Y 56.2645, Z -3.8333, A 0.000, B 0.000, C 0.000 }
gfCNCPoint3[9043] = {X 423.3883, Y 57.1099, Z -3.8333, A 0.000, B 0.000, C 0.000 }
gfCNCPoint3[9044] = {X 423.4886, Y 58.0000, Z -3.8333, A 0.000, B 0.000, C 0.000 }
gfCNCPoint3[9045] = {X 423.4886, Y 58.4511, Z -3.8333, A 0.000, B 0.000, C 0.000 }
gfCNCPoint3[9046] = {X 429.4945, Y 60.7915, Z -3.8333, A 0.000, B 0.000, C 0.000 }
gfCNCPoint3[9047] = {X 458.1787, Y 72.1721, Z -3.8333, A 0.000, B 0.000, C 0.000 }
gfCNCPoint3[9048] = {X 458.1793, Y 63.0385, Z -3.8333, A 0.000, B 0.000, C 0.000 }
gfCNCPoint3[9049] = {X 458.1841, Y 62.9246, Z -3.8333, A 0.000, B 0.000, C 0.000 }
gfCNCPoint3[9050] = {X 458.0122, Y 62.9090, Z -3.8333, A 0.000, B 0.000, C 0.000 }
gfCNCPoint3[9051] = {X 457.8411, Y 62.8860, Z -3.8333, A 0.000, B 0.000, C 0.000 }
gfCNCPoint3[9052] = {X 456.9345, Y 62.6319, Z -3.8333, A 0.000, B 0.000, C 0.000 }
gfCNCPoint3[9053] = {X 456.1124, Y 62.1730, Z -3.8333, A 0.000, B 0.000, C 0.000 }
gfCNCPoint3[9054] = {X 455.4204, Y 61.5346, Z -3.8333, A 0.000, B 0.000, C 0.000 }
gfCNCPoint3[9055] = {X 454.8967, Y 60.7522, Z -3.8333, A 0.000, B 0.000, C 0.000 }
gfCNCPoint3[9056] = {X 454.5704, Y 59.8690, Z -3.8333, A 0.000, B 0.000, C 0.000 }
gfCNCPoint3[9057] = {X 454.4596, Y 58.9340, Z -3.8333, A 0.000, B 0.000, C 0.000 }
gfCNCPoint3[9058] = {X 454.4596, Y 58.0000, Z -3.8333, A 0.000, B 0.000, C 0.000 }
gfCNCPoint3[9059] = {X 454.5599, Y 57.1099, Z -3.8333, A 0.000, B 0.000, C 0.000 }
gfCNCPoint3[9060] = {X 454.8557, Y 56.2645, Z -3.8333, A 0.000, B 0.000, C 0.000 }
gfCNCPoint3[9061] = {X 455.3323, Y 55.5060, Z -3.8333, A 0.000, B 0.000, C 0.000 }
gfCNCPoint3[9062] = {X 455.9656, Y 54.8727, Z -3.8333, A 0.000, B 0.000, C 0.000 }
gfCNCPoint3[9063] = {X 456.7241, Y 54.3961, Z -3.8333, A 0.000, B 0.000, C 0.000 }
gfCNCPoint3[9064] = {X 457.5695, Y 54.1003, Z -3.8333, A 0.000, B 0.000, C 0.000 }
gfCNCPoint3[9065] = {X 458.4596, Y 54.0000, Z -3.8333, A 0.000, B 0.000, C 0.000 }
gfCNCPoint3[9066] = {X 475.0000, Y 54.0000, Z -3.8333, A 0.000, B 0.000, C 0.000 }
gfCNCPoint3[9067] = {X 475.8901, Y 54.1003, Z -3.8333, A 0.000, B 0.000, C 0.000 }
gfCNCPoint3[9068] = {X 476.7355, Y 54.3961, Z -3.8333, A 0.000, B 0.000, C 0.000 }
gfCNCPoint3[9069] = {X 477.4940, Y 54.8727, Z -3.8333, A 0.000, B 0.000, C 0.000 }
gfCNCPoint3[9070] = {X 478.1273, Y 55.5060, Z -3.8333, A 0.000, B 0.000, C 0.000 }
gfCNCPoint3[9071] = {X 478.6039, Y 56.2645, Z -3.8333, A 0.000, B 0.000, C 0.000 }
gfCNCPoint3[9072] = {X 478.8997, Y 57.1099, Z -3.8333, A 0.000, B 0.000, C 0.000 }
gfCNCPoint3[9073] = {X 479.0000, Y 58.0000, Z -3.8333, A 0.000, B 0.000, C 0.000 }
gfCNCPoint3[9074] = {X 478.9999, Y 58.9671, Z -3.8333, A 0.000, B 0.000, C 0.000 }
gfCNCPoint3[9075] = {X 478.9023, Y 59.8127, Z -3.8333, A 0.000, B 0.000, C 0.000 }
gfCNCPoint3[9076] = {X 478.6280, Y 60.6186, Z -3.8333, A 0.000, B 0.000, C 0.000 }
gfCNCPoint3[9077] = {X 478.1894, Y 61.3481, Z -3.8333, A 0.000, B 0.000, C 0.000 }
gfCNCPoint3[9078] = {X 477.6064, Y 61.9683, Z -3.8333, A 0.000, B 0.000, C 0.000 }
gfCNCPoint3[9079] = {X 476.9053, Y 62.4511, Z -3.8333, A 0.000, B 0.000, C 0.000 }
gfCNCPoint3[9080] = {X 476.1180, Y 62.7747, Z -3.8333, A 0.000, B 0.000, C 0.000 }
gfCNCPoint3[9081] = {X 475.2800, Y 62.9243, Z -3.8333, A 0.000, B 0.000, C 0.000 }
gfCNCPoint3[9082] = {X 475.2804, Y 93.0293, Z -3.8333, A 0.000, B 0.000, C 0.000 }
gfCNCPoint3[9083] = {X 475.7877, Y 93.1426, Z -3.8333, A 0.000, B 0.000, C 0.000 }
gfCNCPoint3[9084] = {X 476.2860, Y 93.2904, Z -3.8333, A 0.000, B 0.000, C 0.000 }
gfCNCPoint3[9085] = {X 477.0372, Y 93.6318, Z -3.8333, A 0.000, B 0.000, C 0.000 }
gfCNCPoint3[9086] = {X 477.7017, Y 94.1209, Z -3.8333, A 0.000, B 0.000, C 0.000 }
gfCNCPoint3[9087] = {X 478.2509, Y 94.7368, Z -3.8333, A 0.000, B 0.000, C 0.000 }
gfCNCPoint3[9088] = {X 478.6610, Y 95.4529, Z -3.8333, A 0.000, B 0.000, C 0.000 }
gfCNCPoint3[9089] = {X 478.9143, Y 96.2382, Z -3.8333, A 0.000, B 0.000, C 0.000 }
gfCNCPoint3[9090] = {X 479.0000, Y 97.0589, Z -3.8333, A 0.000, B 0.000, C 0.000 }
gfCNCPoint3[9091] = {X 479.0000, Y 98.0000, Z -3.8333, A 0.000, B 0.000, C 0.000 }
gfCNCPoint3[9092] = {X 478.8997, Y 98.8901, Z -3.8333, A 0.000, B 0.000, C 0.000 }
gfCNCPoint3[9093] = {X 478.6039, Y 99.7355, Z -3.8333, A 0.000, B 0.000, C 0.000 }
gfCNCPoint3[9094] = {X 478.1273, Y 100.4940, Z -3.8333, A 0.000, B 0.000, C 0.000 }
gfCNCPoint3[9095] = {X 477.4940, Y 101.1273, Z -3.8333, A 0.000, B 0.000, C 0.000 }
gfCNCPoint3[9096] = {X 476.7355, Y 101.6039, Z -3.8333, A 0.000, B 0.000, C 0.000 }
gfCNCPoint3[9097] = {X 475.8901, Y 101.8997, Z -3.8333, A 0.000, B 0.000, C 0.000 }
gfCNCPoint3[9098] = {X 475.0000, Y 102.0000, Z -3.8333, A 0.000, B 0.000, C 0.000 }
gfCNCPoint3[9099] = {X 458.4596, Y 102.0000, Z -3.8333, A 0.000, B 0.000, C 0.000 }
gfCNCPoint3[9100] = {X 457.5695, Y 101.8997, Z -3.8333, A 0.000, B 0.000, C 0.000 }
gfCNCPoint3[9101] = {X 456.7241, Y 101.6039, Z -3.8333, A 0.000, B 0.000, C 0.000 }
gfCNCPoint3[9102] = {X 455.9656, Y 101.1273, Z -3.8333, A 0.000, B 0.000, C 0.000 }
gfCNCPoint3[9103] = {X 455.3323, Y 100.4940, Z -3.8333, A 0.000, B 0.000, C 0.000 }
gfCNCPoint3[9104] = {X 454.8557, Y 99.7355, Z -3.8333, A 0.000, B 0.000, C 0.000 }
gfCNCPoint3[9105] = {X 454.5599, Y 98.8901, Z -3.8333, A 0.000, B 0.000, C 0.000 }
gfCNCPoint3[9106] = {X 454.4596, Y 98.0000, Z -3.8333, A 0.000, B 0.000, C 0.000 }
gfCNCPoint3[9107] = {X 454.4596, Y 97.0659, Z -3.8333, A 0.000, B 0.000, C 0.000 }
gfCNCPoint3[9108] = {X 454.5511, Y 96.2154, Z -3.8333, A 0.000, B 0.000, C 0.000 }
gfCNCPoint3[9109] = {X 454.8213, Y 95.4037, Z -3.8333, A 0.000, B 0.000, C 0.000 }
gfCNCPoint3[9110] = {X 455.2580, Y 94.6681, Z -3.8333, A 0.000, B 0.000, C 0.000 }
gfCNCPoint3[9111] = {X 455.8411, Y 94.0422, Z -3.8333, A 0.000, B 0.000, C 0.000 }
gfCNCPoint3[9112] = {X 456.5439, Y 93.5545, Z -3.8333, A 0.000, B 0.000, C 0.000 }
gfCNCPoint3[9113] = {X 457.3344, Y 93.2275, Z -3.8333, A 0.000, B 0.000, C 0.000 }
gfCNCPoint3[9114] = {X 458.1763, Y 93.0760, Z -3.8333, A 0.000, B 0.000, C 0.000 }
gfCNCPoint3[9115] = {X 458.1763, Y 85.3767, Z -3.8333, A 0.000, B 0.000, C 0.000 }
gfCNCPoint3[9116] = {X 445.0138, Y 80.2170, Z -3.8333, A 0.000, B 0.000, C 0.000 }
gfCNCPoint3[9117] = {X 444.8241, Y 80.1411, Z -3.8333, A 0.000, B 0.000, C 0.000 }
gfCNCPoint3[9118] = {X 419.7019, Y 96.4150, Z -3.8333, A 0.000, B 0.000, C 0.000 }
gfCNCPoint3[9119] = {X 419.7067, Y 97.0659, Z -3.8333, A 0.000, B 0.000, C 0.000 }
gfCNCPoint3[9120] = {X 419.7067, Y 98.0000, Z -3.8333, A 0.000, B 0.000, C 0.000 }
gfCNCPoint3[9121] = {X 419.6064, Y 98.8901, Z -3.8333, A 0.000, B 0.000, C 0.000 }
gfCNCPoint3[9122] = {X 419.3106, Y 99.7355, Z -3.8333, A 0.000, B 0.000, C 0.000 }
gfCNCPoint3[9123] = {X 418.8340, Y 100.4940, Z -3.8333, A 0.000, B 0.000, C 0.000 }
gfCNCPoint3[9124] = {X 418.2007, Y 101.1273, Z -3.8333, A 0.000, B 0.000, C 0.000 }
gfCNCPoint3[9125] = {X 417.4422, Y 101.6039, Z -3.8333, A 0.000, B 0.000, C 0.000 }
gfCNCPoint3[9126] = {X 416.5968, Y 101.8997, Z -3.8333, A 0.000, B 0.000, C 0.000 }
gfCNCPoint3[9127] = {X 415.7067, Y 102.0000, Z -3.8333, A 0.000, B 0.000, C 0.000 }
gfCNCPoint3[9128] = {X 396.4059, Y 102.0000, Z -3.8333, A 0.000, B 0.000, C 0.000 }
gfCNCPoint3[9129] = {X 395.5159, Y 101.8997, Z -3.8333, A 0.000, B 0.000, C 0.000 }
gfCNCPoint3[9130] = {X 394.6704, Y 101.6039, Z -3.8333, A 0.000, B 0.000, C 0.000 }
gfCNCPoint3[9131] = {X 393.9120, Y 101.1273, Z -3.8333, A 0.000, B 0.000, C 0.000 }
gfCNCPoint3[9132] = {X 393.2786, Y 100.4940, Z -3.8333, A 0.000, B 0.000, C 0.000 }
gfCNCPoint3[9133] = {X 392.8021, Y 99.7355, Z -3.8333, A 0.000, B 0.000, C 0.000 }
gfCNCPoint3[9134] = {X 392.5062, Y 98.8901, Z -3.8333, A 0.000, B 0.000, C 0.000 }
gfCNCPoint3[9135] = {X 392.4059, Y 98.0000, Z -3.8333, A 0.000, B 0.000, C 0.000 }
gfCNCPoint3[9136] = {X 392.4059, Y 97.0659, Z -3.8333, A 0.000, B 0.000, C 0.000 }
gfCNCPoint3[9137] = {X 392.5074, Y 96.1706, Z -3.8333, A 0.000, B 0.000, C 0.000 }
gfCNCPoint3[9138] = {X 392.8067, Y 95.3207, Z -3.8333, A 0.000, B 0.000, C 0.000 }
gfCNCPoint3[9139] = {X 393.2887, Y 94.5594, Z -3.8333, A 0.000, B 0.000, C 0.000 }
gfCNCPoint3[9140] = {X 393.9288, Y 93.9253, Z -3.8333, A 0.000, B 0.000, C 0.000 }
gfCNCPoint3[9141] = {X 394.6946, Y 93.4505, Z -3.8333, A 0.000, B 0.000, C 0.000 }
gfCNCPoint3[9142] = {X 395.5473, Y 93.1592, Z -3.8333, A 0.000, B 0.000, C 0.000 }
gfCNCPoint3[9143] = {X 396.4435, Y 93.0661, Z -3.8333, A 0.000, B 0.000, C 0.000 }
gfCNCPoint3[9144] = {X 397.3897, Y 93.0222, Z -3.8333, A 0.000, B 0.000, C 0.000 }
gfCNCPoint3[9145] = {X 398.3327, Y 92.9322, Z -3.8333, A 0.000, B 0.000, C 0.000 }
gfCNCPoint3[9146] = {X 399.0538, Y 92.7577, Z -3.8333, A 0.000, B 0.000, C 0.000 }
gfCNCPoint3[9147] = {X 399.7177, Y 92.4265, Z -3.8333, A 0.000, B 0.000, C 0.000 }
gfCNCPoint3[9148] = {X 405.3925, Y 88.7698, Z -3.8333, A 0.000, B 0.000, C 0.000 }
gfCNCPoint3[9149] = {X 413.9653, Y 83.2882, Z -3.8333, A 0.000, B 0.000, C 0.000 }
gfCNCPoint3[9150] = {X 411.7673, Y 79.8508, Z -3.8333, A 0.000, B 0.000, C 0.000 }
gfCNCPoint3[9151] = {X 411.7673, Y 79.8508, Z -0.8333, A 0.000, B 0.000, C 0.000 }
gfCNCPoint3[9152] = {X 411.7673, Y 79.8508, Z 11.0000, A 0.000, B 0.000, C 0.000 }
gfCNCPoint3[9153] = {X 466.3105, Y 28.5935, Z 11.0000, A 0.000, B 0.000, C 0.000 }
gfCNCPoint3[9154] = {X 466.3105, Y 28.5935, Z -0.8333, A 0.000, B 0.000, C 0.000 }
gfCNCPoint3[9155] = {X 466.3105, Y 28.5935, Z -3.8333, A 0.000, B 0.000, C 0.000 }
gfCNCPoint3[9156] = {X 462.2305, Y 28.5935, Z -3.8333, A 0.000, B 0.000, C 0.000 }
gfCNCPoint3[9157] = {X 462.2307, Y 40.9133, Z -3.8333, A 0.000, B 0.000, C 0.000 }
gfCNCPoint3[9158] = {X 462.2394, Y 40.9203, Z -3.8333, A 0.000, B 0.000, C 0.000 }
gfCNCPoint3[9159] = {X 462.8743, Y 41.5908, Z -3.8333, A 0.000, B 0.000, C 0.000 }
gfCNCPoint3[9160] = {X 463.3522, Y 42.3809, Z -3.8333, A 0.000, B 0.000, C 0.000 }
gfCNCPoint3[9161] = {X 463.6512, Y 43.2545, Z -3.8333, A 0.000, B 0.000, C 0.000 }
gfCNCPoint3[9162] = {X 463.7578, Y 44.1718, Z -3.8333, A 0.000, B 0.000, C 0.000 }
gfCNCPoint3[9163] = {X 463.7579, Y 45.0000, Z -3.8333, A 0.000, B 0.000, C 0.000 }
gfCNCPoint3[9164] = {X 463.6496, Y 45.9613, Z -3.8333, A 0.000, B 0.000, C 0.000 }
gfCNCPoint3[9165] = {X 463.3301, Y 46.8744, Z -3.8333, A 0.000, B 0.000, C 0.000 }
gfCNCPoint3[9166] = {X 462.8155, Y 47.6935, Z -3.8333, A 0.000, B 0.000, C 0.000 }
gfCNCPoint3[9167] = {X 462.1314, Y 48.3775, Z -3.8333, A 0.000, B 0.000, C 0.000 }
gfCNCPoint3[9168] = {X 461.3123, Y 48.8922, Z -3.8333, A 0.000, B 0.000, C 0.000 }
gfCNCPoint3[9169] = {X 460.3992, Y 49.2117, Z -3.8333, A 0.000, B 0.000, C 0.000 }
gfCNCPoint3[9170] = {X 459.4379, Y 49.3200, Z -3.8333, A 0.000, B 0.000, C 0.000 }
gfCNCPoint3[9171] = {X 452.9945, Y 49.3200, Z -3.8333, A 0.000, B 0.000, C 0.000 }
gfCNCPoint3[9172] = {X 452.0380, Y 49.2128, Z -3.8333, A 0.000, B 0.000, C 0.000 }
gfCNCPoint3[9173] = {X 451.1291, Y 48.8965, Z -3.8333, A 0.000, B 0.000, C 0.000 }
gfCNCPoint3[9174] = {X 450.3127, Y 48.3868, Z -3.8333, A 0.000, B 0.000, C 0.000 }
gfCNCPoint3[9175] = {X 449.6294, Y 47.7091, Z -3.8333, A 0.000, B 0.000, C 0.000 }
gfCNCPoint3[9176] = {X 449.1132, Y 46.8968, Z -3.8333, A 0.000, B 0.000, C 0.000 }
gfCNCPoint3[9177] = {X 448.7896, Y 45.9905, Z -3.8333, A 0.000, B 0.000, C 0.000 }
gfCNCPoint3[9178] = {X 448.6746, Y 45.0349, Z -3.8333, A 0.000, B 0.000, C 0.000 }
gfCNCPoint3[9179] = {X 448.6749, Y 44.1494, Z -3.8333, A 0.000, B 0.000, C 0.000 }
gfCNCPoint3[9180] = {X 448.7853, Y 43.2364, Z -3.8333, A 0.000, B 0.000, C 0.000 }
gfCNCPoint3[9181] = {X 449.0865, Y 42.3675, Z -3.8333, A 0.000, B 0.000, C 0.000 }
gfCNCPoint3[9182] = {X 449.5648, Y 41.5821, Z -3.8333, A 0.000, B 0.000, C 0.000 }
gfCNCPoint3[9183] = {X 450.1984, Y 40.9157, Z -3.8333, A 0.000, B 0.000, C 0.000 }
gfCNCPoint3[9184] = {X 450.1984, Y 34.4738, Z -3.8333, A 0.000, B 0.000, C 0.000 }
gfCNCPoint3[9185] = {X 447.4743, Y 34.4738, Z -3.8333, A 0.000, B 0.000, C 0.000 }
gfCNCPoint3[9186] = {X 443.1895, Y 42.8163, Z -3.8333, A 0.000, B 0.000, C 0.000 }
gfCNCPoint3[9187] = {X 443.1945, Y 42.8300, Z -3.8333, A 0.000, B 0.000, C 0.000 }
gfCNCPoint3[9188] = {X 443.3605, Y 43.4912, Z -3.8333, A 0.000, B 0.000, C 0.000 }
gfCNCPoint3[9189] = {X 443.4203, Y 44.1703, Z -3.8333, A 0.000, B 0.000, C 0.000 }
gfCNCPoint3[9190] = {X 443.4205, Y 45.0000, Z -3.8333, A 0.000, B 0.000, C 0.000 }
gfCNCPoint3[9191] = {X 443.3122, Y 45.9613, Z -3.8333, A 0.000, B 0.000, C 0.000 }
gfCNCPoint3[9192] = {X 442.9927, Y 46.8744, Z -3.8333, A 0.000, B 0.000, C 0.000 }
gfCNCPoint3[9193] = {X 442.4780, Y 47.6935, Z -3.8333, A 0.000, B 0.000, C 0.000 }
gfCNCPoint3[9194] = {X 441.7939, Y 48.3775, Z -3.8333, A 0.000, B 0.000, C 0.000 }
gfCNCPoint3[9195] = {X 440.9748, Y 48.8922, Z -3.8333, A 0.000, B 0.000, C 0.000 }
gfCNCPoint3[9196] = {X 440.0618, Y 49.2117, Z -3.8333, A 0.000, B 0.000, C 0.000 }
gfCNCPoint3[9197] = {X 439.1005, Y 49.3200, Z -3.8333, A 0.000, B 0.000, C 0.000 }
gfCNCPoint3[9198] = {X 432.5144, Y 49.3200, Z -3.8333, A 0.000, B 0.000, C 0.000 }
gfCNCPoint3[9199] = {X 431.5531, Y 49.2117, Z -3.8333, A 0.000, B 0.000, C 0.000 }
gfCNCPoint3[9200] = {X 430.6401, Y 48.8922, Z -3.8333, A 0.000, B 0.000, C 0.000 }
gfCNCPoint3[9201] = {X 429.8210, Y 48.3775, Z -3.8333, A 0.000, B 0.000, C 0.000 }
gfCNCPoint3[9202] = {X 429.1369, Y 47.6935, Z -3.8333, A 0.000, B 0.000, C 0.000 }
gfCNCPoint3[9203] = {X 428.6223, Y 46.8745, Z -3.8333, A 0.000, B 0.000, C 0.000 }
gfCNCPoint3[9204] = {X 428.3027, Y 45.9614, Z -3.8333, A 0.000, B 0.000, C 0.000 }
gfCNCPoint3[9205] = {X 428.1944, Y 45.0001, Z -3.8333, A 0.000, B 0.000, C 0.000 }
gfCNCPoint3[9206] = {X 428.1948, Y 44.1494, Z -3.8333, A 0.000, B 0.000, C 0.000 }
gfCNCPoint3[9207] = {X 428.2925, Y 43.2935, Z -3.8333, A 0.000, B 0.000, C 0.000 }
gfCNCPoint3[9208] = {X 428.5580, Y 42.4740, Z -3.8333, A 0.000, B 0.000, C 0.000 }
gfCNCPoint3[9209] = {X 428.9809, Y 41.7236, Z -3.8333, A 0.000, B 0.000, C 0.000 }
gfCNCPoint3[9210] = {X 429.5442, Y 41.0719, Z -3.8333, A 0.000, B 0.000, C 0.000 }
gfCNCPoint3[9211] = {X 430.2256, Y 40.5449, Z -3.8333, A 0.000, B 0.000, C 0.000 }
gfCNCPoint3[9212] = {X 430.9981, Y 40.1637, Z -3.8333, A 0.000, B 0.000, C 0.000 }
gfCNCPoint3[9213] = {X 434.9872, Y 32.3554, Z -3.8333, A 0.000, B 0.000, C 0.000 }
gfCNCPoint3[9214] = {X 433.8173, Y 31.5689, Z -3.8333, A 0.000, B 0.000, C 0.000 }
gfCNCPoint3[9215] = {X 432.7542, Y 30.6430, Z -3.8333, A 0.000, B 0.000, C 0.000 }
gfCNCPoint3[9216] = {X 431.8144, Y 29.5923, Z -3.8333, A 0.000, B 0.000, C 0.000 }
gfCNCPoint3[9217] = {X 431.0125, Y 28.4329, Z -3.8333, A 0.000, B 0.000, C 0.000 }
gfCNCPoint3[9218] = {X 430.3608, Y 27.1828, Z -3.8333, A 0.000, B 0.000, C 0.000 }
gfCNCPoint3[9219] = {X 429.8696, Y 25.8615, Z -3.8333, A 0.000, B 0.000, C 0.000 }
gfCNCPoint3[9220] = {X 429.4505, Y 24.0500, Z -3.8333, A 0.000, B 0.000, C 0.000 }
gfCNCPoint3[9221] = {X 429.2369, Y 22.2029, Z -3.8333, A 0.000, B 0.000, C 0.000 }
gfCNCPoint3[9222] = {X 429.2315, Y 20.3436, Z -3.8333, A 0.000, B 0.000, C 0.000 }
gfCNCPoint3[9223] = {X 429.4344, Y 18.4953, Z -3.8333, A 0.000, B 0.000, C 0.000 }
gfCNCPoint3[9224] = {X 429.8430, Y 16.6814, Z -3.8333, A 0.000, B 0.000, C 0.000 }
gfCNCPoint3[9225] = {X 430.3646, Y 15.2116, Z -3.8333, A 0.000, B 0.000, C 0.000 }
gfCNCPoint3[9226] = {X 431.0755, Y 13.8234, Z -3.8333, A 0.000, B 0.000, C 0.000 }
gfCNCPoint3[9227] = {X 431.9633, Y 12.5412, Z -3.8333, A 0.000, B 0.000, C 0.000 }
gfCNCPoint3[9228] = {X 433.0126, Y 11.3873, Z -3.8333, A 0.000, B 0.000, C 0.000 }
gfCNCPoint3[9229] = {X 434.2049, Y 10.3820, Z -3.8333, A 0.000, B 0.000, C 0.000 }
gfCNCPoint3[9230] = {X 435.5194, Y 9.5427, Z -3.8333, A 0.000, B 0.000, C 0.000 }
gfCNCPoint3[9231] = {X 436.9332, Y 8.8842, Z -3.8333, A 0.000, B 0.000, C 0.000 }
gfCNCPoint3[9232] = {X 438.4215, Y 8.4180, Z -3.8333, A 0.000, B 0.000, C 0.000 }
gfCNCPoint3[9233] = {X 440.0467, Y 8.1095, Z -3.8333, A 0.000, B 0.000, C 0.000 }
gfCNCPoint3[9234] = {X 441.6910, Y 7.9281, Z -3.8333, A 0.000, B 0.000, C 0.000 }
gfCNCPoint3[9235] = {X 443.3443, Y 7.8749, Z -3.8333, A 0.000, B 0.000, C 0.000 }
gfCNCPoint3[9236] = {X 444.0357, Y 7.8709, Z -3.8333, A 0.000, B 0.000, C 0.000 }
gfCNCPoint3[9237] = {X 459.4467, Y 7.8709, Z -3.8333, A 0.000, B 0.000, C 0.000 }
gfCNCPoint3[9238] = {X 460.4060, Y 7.9790, Z -3.8333, A 0.000, B 0.000, C 0.000 }
gfCNCPoint3[9239] = {X 461.3173, Y 8.2979, Z -3.8333, A 0.000, B 0.000, C 0.000 }
gfCNCPoint3[9240] = {X 462.1347, Y 8.8115, Z -3.8333, A 0.000, B 0.000, C 0.000 }
gfCNCPoint3[9241] = {X 462.8174, Y 9.4941, Z -3.8333, A 0.000, B 0.000, C 0.000 }
gfCNCPoint3[9242] = {X 463.3310, Y 10.3116, Z -3.8333, A 0.000, B 0.000, C 0.000 }
gfCNCPoint3[9243] = {X 463.6498, Y 11.2228, Z -3.8333, A 0.000, B 0.000, C 0.000 }
gfCNCPoint3[9244] = {X 463.7579, Y 12.1822, Z -3.8333, A 0.000, B 0.000, C 0.000 }
gfCNCPoint3[9245] = {X 463.7579, Y 12.9782, Z -3.8333, A 0.000, B 0.000, C 0.000 }
gfCNCPoint3[9246] = {X 463.6565, Y 13.9081, Z -3.8333, A 0.000, B 0.000, C 0.000 }
gfCNCPoint3[9247] = {X 463.3574, Y 14.7943, Z -3.8333, A 0.000, B 0.000, C 0.000 }
gfCNCPoint3[9248] = {X 462.8744, Y 15.5954, Z -3.8333, A 0.000, B 0.000, C 0.000 }
gfCNCPoint3[9249] = {X 462.2303, Y 16.2738, Z -3.8333, A 0.000, B 0.000, C 0.000 }
gfCNCPoint3[9250] = {X 462.2305, Y 28.5935, Z -3.8333, A 0.000, B 0.000, C 0.000 }
gfCNCPoint3[9251] = {X 466.2305, Y 28.5935, Z -3.8333, A 0.000, B 0.000, C 0.000 }
gfCNCPoint3[9252] = {X 462.1505, Y 28.5935, Z -3.8333, A 0.000, B 0.000, C 0.000 }
gfCNCPoint3[9253] = {X 462.1507, Y 40.9513, Z -3.8333, A 0.000, B 0.000, C 0.000 }
gfCNCPoint3[9254] = {X 462.1882, Y 40.9818, Z -3.8333, A 0.000, B 0.000, C 0.000 }
gfCNCPoint3[9255] = {X 462.8111, Y 41.6398, Z -3.8333, A 0.000, B 0.000, C 0.000 }
gfCNCPoint3[9256] = {X 463.2799, Y 42.4152, Z -3.8333, A 0.000, B 0.000, C 0.000 }
gfCNCPoint3[9257] = {X 463.5733, Y 43.2724, Z -3.8333, A 0.000, B 0.000, C 0.000 }
gfCNCPoint3[9258] = {X 463.6778, Y 44.1724, Z -3.8333, A 0.000, B 0.000, C 0.000 }
gfCNCPoint3[9259] = {X 463.6779, Y 45.0000, Z -3.8333, A 0.000, B 0.000, C 0.000 }
gfCNCPoint3[9260] = {X 463.5716, Y 45.9435, Z -3.8333, A 0.000, B 0.000, C 0.000 }
gfCNCPoint3[9261] = {X 463.2580, Y 46.8397, Z -3.8333, A 0.000, B 0.000, C 0.000 }
gfCNCPoint3[9262] = {X 462.7529, Y 47.6436, Z -3.8333, A 0.000, B 0.000, C 0.000 }
gfCNCPoint3[9263] = {X 462.0815, Y 48.3150, Z -3.8333, A 0.000, B 0.000, C 0.000 }
gfCNCPoint3[9264] = {X 461.2776, Y 48.8201, Z -3.8333, A 0.000, B 0.000, C 0.000 }
gfCNCPoint3[9265] = {X 460.3814, Y 49.1337, Z -3.8333, A 0.000, B 0.000, C 0.000 }
gfCNCPoint3[9266] = {X 459.4379, Y 49.2400, Z -3.8333, A 0.000, B 0.000, C 0.000 }
gfCNCPoint3[9267] = {X 452.9945, Y 49.2400, Z -3.8333, A 0.000, B 0.000, C 0.000 }
gfCNCPoint3[9268] = {X 452.0558, Y 49.1348, Z -3.8333, A 0.000, B 0.000, C 0.000 }
gfCNCPoint3[9269] = {X 451.1636, Y 48.8243, Z -3.8333, A 0.000, B 0.000, C 0.000 }
gfCNCPoint3[9270] = {X 450.3624, Y 48.3241, Z -3.8333, A 0.000, B 0.000, C 0.000 }
gfCNCPoint3[9271] = {X 449.6918, Y 47.6589, Z -3.8333, A 0.000, B 0.000, C 0.000 }
gfCNCPoint3[9272] = {X 449.1851, Y 46.8617, Z -3.8333, A 0.000, B 0.000, C 0.000 }
gfCNCPoint3[9273] = {X 448.8674, Y 45.9721, Z -3.8333, A 0.000, B 0.000, C 0.000 }
gfCNCPoint3[9274] = {X 448.7546, Y 45.0343, Z -3.8333, A 0.000, B 0.000, C 0.000 }
gfCNCPoint3[9275] = {X 448.7549, Y 44.1505, Z -3.8333, A 0.000, B 0.000, C 0.000 }
gfCNCPoint3[9276] = {X 448.8654, Y 43.2454, Z -3.8333, A 0.000, B 0.000, C 0.000 }
gfCNCPoint3[9277] = {X 449.1668, Y 42.3850, Z -3.8333, A 0.000, B 0.000, C 0.000 }
gfCNCPoint3[9278] = {X 449.6452, Y 41.6088, Z -3.8333, A 0.000, B 0.000, C 0.000 }
gfCNCPoint3[9279] = {X 450.2784, Y 40.9529, Z -3.8333, A 0.000, B 0.000, C 0.000 }
gfCNCPoint3[9280] = {X 450.2784, Y 34.3938, Z -3.8333, A 0.000, B 0.000, C 0.000 }
gfCNCPoint3[9281] = {X 447.4255, Y 34.3938, Z -3.8333, A 0.000, B 0.000, C 0.000 }
gfCNCPoint3[9282] = {X 443.1023, Y 42.8110, Z -3.8333, A 0.000, B 0.000, C 0.000 }
gfCNCPoint3[9283] = {X 443.1191, Y 42.8565, Z -3.8333, A 0.000, B 0.000, C 0.000 }
gfCNCPoint3[9284] = {X 443.2817, Y 43.5050, Z -3.8333, A 0.000, B 0.000, C 0.000 }
gfCNCPoint3[9285] = {X 443.3403, Y 44.1710, Z -3.8333, A 0.000, B 0.000, C 0.000 }
gfCNCPoint3[9286] = {X 443.3405, Y 45.0000, Z -3.8333, A 0.000, B 0.000, C 0.000 }
gfCNCPoint3[9287] = {X 443.2342, Y 45.9435, Z -3.8333, A 0.000, B 0.000, C 0.000 }
gfCNCPoint3[9288] = {X 442.9206, Y 46.8397, Z -3.8333, A 0.000, B 0.000, C 0.000 }
gfCNCPoint3[9289] = {X 442.4154, Y 47.6436, Z -3.8333, A 0.000, B 0.000, C 0.000 }
gfCNCPoint3[9290] = {X 441.7441, Y 48.3150, Z -3.8333, A 0.000, B 0.000, C 0.000 }
gfCNCPoint3[9291] = {X 440.9401, Y 48.8201, Z -3.8333, A 0.000, B 0.000, C 0.000 }
gfCNCPoint3[9292] = {X 440.0440, Y 49.1337, Z -3.8333, A 0.000, B 0.000, C 0.000 }
gfCNCPoint3[9293] = {X 439.1005, Y 49.2400, Z -3.8333, A 0.000, B 0.000, C 0.000 }
gfCNCPoint3[9294] = {X 432.5144, Y 49.2400, Z -3.8333, A 0.000, B 0.000, C 0.000 }
gfCNCPoint3[9295] = {X 431.5709, Y 49.1337, Z -3.8333, A 0.000, B 0.000, C 0.000 }
gfCNCPoint3[9296] = {X 430.6748, Y 48.8201, Z -3.8333, A 0.000, B 0.000, C 0.000 }
gfCNCPoint3[9297] = {X 429.8708, Y 48.3150, Z -3.8333, A 0.000, B 0.000, C 0.000 }
gfCNCPoint3[9298] = {X 429.1995, Y 47.6436, Z -3.8333, A 0.000, B 0.000, C 0.000 }
gfCNCPoint3[9299] = {X 428.6943, Y 46.8397, Z -3.8333, A 0.000, B 0.000, C 0.000 }
gfCNCPoint3[9300] = {X 428.3807, Y 45.9436, Z -3.8333, A 0.000, B 0.000, C 0.000 }
gfCNCPoint3[9301] = {X 428.2744, Y 45.0001, Z -3.8333, A 0.000, B 0.000, C 0.000 }
gfCNCPoint3[9302] = {X 428.2748, Y 44.1505, Z -3.8333, A 0.000, B 0.000, C 0.000 }
gfCNCPoint3[9303] = {X 428.3718, Y 43.3054, Z -3.8333, A 0.000, B 0.000, C 0.000 }
gfCNCPoint3[9304] = {X 428.6354, Y 42.4967, Z -3.8333, A 0.000, B 0.000, C 0.000 }
gfCNCPoint3[9305] = {X 429.0552, Y 41.7570, Z -3.8333, A 0.000, B 0.000, C 0.000 }
gfCNCPoint3[9306] = {X 429.6142, Y 41.1158, Z -3.8333, A 0.000, B 0.000, C 0.000 }
gfCNCPoint3[9307] = {X 430.2899, Y 40.5992, Z -3.8333, A 0.000, B 0.000, C 0.000 }
gfCNCPoint3[9308] = {X 431.0551, Y 40.2278, Z -3.8333, A 0.000, B 0.000, C 0.000 }
gfCNCPoint3[9309] = {X 435.0929, Y 32.3243, Z -3.8333, A 0.000, B 0.000, C 0.000 }
gfCNCPoint3[9310] = {X 433.9160, Y 31.5435, Z -3.8333, A 0.000, B 0.000, C 0.000 }
gfCNCPoint3[9311] = {X 432.8463, Y 30.6214, Z -3.8333, A 0.000, B 0.000, C 0.000 }
gfCNCPoint3[9312] = {X 431.9007, Y 29.5724, Z -3.8333, A 0.000, B 0.000, C 0.000 }
gfCNCPoint3[9313] = {X 431.0940, Y 28.4131, Z -3.8333, A 0.000, B 0.000, C 0.000 }
gfCNCPoint3[9314] = {X 430.4391, Y 27.1619, Z -3.8333, A 0.000, B 0.000, C 0.000 }
gfCNCPoint3[9315] = {X 429.9462, Y 25.8383, Z -3.8333, A 0.000, B 0.000, C 0.000 }
gfCNCPoint3[9316] = {X 429.5292, Y 24.0357, Z -3.8333, A 0.000, B 0.000, C 0.000 }
gfCNCPoint3[9317] = {X 429.3167, Y 22.1977, Z -3.8333, A 0.000, B 0.000, C 0.000 }
gfCNCPoint3[9318] = {X 429.3114, Y 20.3475, Z -3.8333, A 0.000, B 0.000, C 0.000 }
gfCNCPoint3[9319] = {X 429.5133, Y 18.5083, Z -3.8333, A 0.000, B 0.000, C 0.000 }
gfCNCPoint3[9320] = {X 429.9200, Y 16.7033, Z -3.8333, A 0.000, B 0.000, C 0.000 }
gfCNCPoint3[9321] = {X 430.4380, Y 15.2434, Z -3.8333, A 0.000, B 0.000, C 0.000 }
gfCNCPoint3[9322] = {X 431.1440, Y 13.8646, Z -3.8333, A 0.000, B 0.000, C 0.000 }
gfCNCPoint3[9323] = {X 432.0258, Y 12.5911, Z -3.8333, A 0.000, B 0.000, C 0.000 }
gfCNCPoint3[9324] = {X 433.0680, Y 11.4450, Z -3.8333, A 0.000, B 0.000, C 0.000 }
gfCNCPoint3[9325] = {X 434.2522, Y 10.4464, Z -3.8333, A 0.000, B 0.000, C 0.000 }
gfCNCPoint3[9326] = {X 435.5579, Y 9.6129, Z -3.8333, A 0.000, B 0.000, C 0.000 }
gfCNCPoint3[9327] = {X 436.9621, Y 8.9588, Z -3.8333, A 0.000, B 0.000, C 0.000 }
gfCNCPoint3[9328] = {X 438.4404, Y 8.4958, Z -3.8333, A 0.000, B 0.000, C 0.000 }
gfCNCPoint3[9329] = {X 440.0593, Y 8.1885, Z -3.8333, A 0.000, B 0.000, C 0.000 }
gfCNCPoint3[9330] = {X 441.6973, Y 8.0078, Z -3.8333, A 0.000, B 0.000, C 0.000 }
gfCNCPoint3[9331] = {X 443.3443, Y 7.9550, Z -3.8333, A 0.000, B 0.000, C 0.000 }
gfCNCPoint3[9332] = {X 444.0360, Y 7.9509, Z -3.8333, A 0.000, B 0.000, C 0.000 }
gfCNCPoint3[9333] = {X 459.4467, Y 7.9509, Z -3.8333, A 0.000, B 0.000, C 0.000 }
gfCNCPoint3[9334] = {X 460.3882, Y 8.0570, Z -3.8333, A 0.000, B 0.000, C 0.000 }
gfCNCPoint3[9335] = {X 461.2825, Y 8.3699, Z -3.8333, A 0.000, B 0.000, C 0.000 }
gfCNCPoint3[9336] = {X 462.0848, Y 8.8740, Z -3.8333, A 0.000, B 0.000, C 0.000 }
gfCNCPoint3[9337] = {X 462.7548, Y 9.5440, Z -3.8333, A 0.000, B 0.000, C 0.000 }
gfCNCPoint3[9338] = {X 463.2589, Y 10.3463, Z -3.8333, A 0.000, B 0.000, C 0.000 }
gfCNCPoint3[9339] = {X 463.5719, Y 11.2406, Z -3.8333, A 0.000, B 0.000, C 0.000 }
gfCNCPoint3[9340] = {X 463.6779, Y 12.1822, Z -3.8333, A 0.000, B 0.000, C 0.000 }
gfCNCPoint3[9341] = {X 463.6779, Y 12.9781, Z -3.8333, A 0.000, B 0.000, C 0.000 }
gfCNCPoint3[9342] = {X 463.5764, Y 13.8998, Z -3.8333, A 0.000, B 0.000, C 0.000 }
gfCNCPoint3[9343] = {X 463.2770, Y 14.7774, Z -3.8333, A 0.000, B 0.000, C 0.000 }
gfCNCPoint3[9344] = {X 462.7939, Y 15.5689, Z -3.8333, A 0.000, B 0.000, C 0.000 }
gfCNCPoint3[9345] = {X 462.1503, Y 16.2365, Z -3.8333, A 0.000, B 0.000, C 0.000 }
gfCNCPoint3[9346] = {X 462.1505, Y 28.5935, Z -3.8333, A 0.000, B 0.000, C 0.000 }
gfCNCPoint3[9347] = {X 466.1505, Y 28.5935, Z -3.8333, A 0.000, B 0.000, C 0.000 }
gfCNCPoint3[9348] = {X 462.0705, Y 28.5935, Z -3.8333, A 0.000, B 0.000, C 0.000 }
gfCNCPoint3[9349] = {X 462.0707, Y 40.9894, Z -3.8333, A 0.000, B 0.000, C 0.000 }
gfCNCPoint3[9350] = {X 462.1370, Y 41.0432, Z -3.8333, A 0.000, B 0.000, C 0.000 }
gfCNCPoint3[9351] = {X 462.7478, Y 41.6888, Z -3.8333, A 0.000, B 0.000, C 0.000 }
gfCNCPoint3[9352] = {X 463.2076, Y 42.4494, Z -3.8333, A 0.000, B 0.000, C 0.000 }
gfCNCPoint3[9353] = {X 463.4953, Y 43.2903, Z -3.8333, A 0.000, B 0.000, C 0.000 }
gfCNCPoint3[9354] = {X 463.5978, Y 44.1731, Z -3.8333, A 0.000, B 0.000, C 0.000 }
gfCNCPoint3[9355] = {X 463.5979, Y 45.0000, Z -3.8333, A 0.000, B 0.000, C 0.000 }
gfCNCPoint3[9356] = {X 463.4936, Y 45.9257, Z -3.8333, A 0.000, B 0.000, C 0.000 }
gfCNCPoint3[9357] = {X 463.1860, Y 46.8050, Z -3.8333, A 0.000, B 0.000, C 0.000 }
gfCNCPoint3[9358] = {X 462.6904, Y 47.5937, Z -3.8333, A 0.000, B 0.000, C 0.000 }
gfCNCPoint3[9359] = {X 462.0317, Y 48.2524, Z -3.8333, A 0.000, B 0.000, C 0.000 }
gfCNCPoint3[9360] = {X 461.2429, Y 48.7480, Z -3.8333, A 0.000, B 0.000, C 0.000 }
gfCNCPoint3[9361] = {X 460.3636, Y 49.0557, Z -3.8333, A 0.000, B 0.000, C 0.000 }
gfCNCPoint3[9362] = {X 459.4379, Y 49.1600, Z -3.8333, A 0.000, B 0.000, C 0.000 }
gfCNCPoint3[9363] = {X 452.9945, Y 49.1600, Z -3.8333, A 0.000, B 0.000, C 0.000 }
gfCNCPoint3[9364] = {X 452.0735, Y 49.0568, Z -3.8333, A 0.000, B 0.000, C 0.000 }
gfCNCPoint3[9365] = {X 451.1982, Y 48.7522, Z -3.8333, A 0.000, B 0.000, C 0.000 }
gfCNCPoint3[9366] = {X 450.4120, Y 48.2614, Z -3.8333, A 0.000, B 0.000, C 0.000 }
gfCNCPoint3[9367] = {X 449.7541, Y 47.6087, Z -3.8333, A 0.000, B 0.000, C 0.000 }
gfCNCPoint3[9368] = {X 449.2569, Y 46.8266, Z -3.8333, A 0.000, B 0.000, C 0.000 }
gfCNCPoint3[9369] = {X 448.9453, Y 45.9538, Z -3.8333, A 0.000, B 0.000, C 0.000 }
gfCNCPoint3[9370] = {X 448.8346, Y 45.0336, Z -3.8333, A 0.000, B 0.000, C 0.000 }
gfCNCPoint3[9371] = {X 448.8349, Y 44.1516, Z -3.8333, A 0.000, B 0.000, C 0.000 }
gfCNCPoint3[9372] = {X 448.9454, Y 43.2545, Z -3.8333, A 0.000, B 0.000, C 0.000 }
gfCNCPoint3[9373] = {X 449.2471, Y 42.4026, Z -3.8333, A 0.000, B 0.000, C 0.000 }
gfCNCPoint3[9374] = {X 449.7256, Y 41.6358, Z -3.8333, A 0.000, B 0.000, C 0.000 }
gfCNCPoint3[9375] = {X 450.3584, Y 40.9906, Z -3.8333, A 0.000, B 0.000, C 0.000 }
gfCNCPoint3[9376] = {X 450.3584, Y 34.3138, Z -3.8333, A 0.000, B 0.000, C 0.000 }
gfCNCPoint3[9377] = {X 447.3766, Y 34.3138, Z -3.8333, A 0.000, B 0.000, C 0.000 }
gfCNCPoint3[9378] = {X 443.0151, Y 42.8057, Z -3.8333, A 0.000, B 0.000, C 0.000 }
gfCNCPoint3[9379] = {X 443.0436, Y 42.8831, Z -3.8333, A 0.000, B 0.000, C 0.000 }
gfCNCPoint3[9380] = {X 443.2029, Y 43.5189, Z -3.8333, A 0.000, B 0.000, C 0.000 }
gfCNCPoint3[9381] = {X 443.2603, Y 44.1717, Z -3.8333, A 0.000, B 0.000, C 0.000 }
gfCNCPoint3[9382] = {X 443.2605, Y 45.0000, Z -3.8333, A 0.000, B 0.000, C 0.000 }
gfCNCPoint3[9383] = {X 443.1562, Y 45.9257, Z -3.8333, A 0.000, B 0.000, C 0.000 }
gfCNCPoint3[9384] = {X 442.8485, Y 46.8050, Z -3.8333, A 0.000, B 0.000, C 0.000 }
gfCNCPoint3[9385] = {X 442.3529, Y 47.5937, Z -3.8333, A 0.000, B 0.000, C 0.000 }
gfCNCPoint3[9386] = {X 441.6942, Y 48.2524, Z -3.8333, A 0.000, B 0.000, C 0.000 }
gfCNCPoint3[9387] = {X 440.9054, Y 48.7480, Z -3.8333, A 0.000, B 0.000, C 0.000 }
gfCNCPoint3[9388] = {X 440.0262, Y 49.0557, Z -3.8333, A 0.000, B 0.000, C 0.000 }
gfCNCPoint3[9389] = {X 439.1005, Y 49.1600, Z -3.8333, A 0.000, B 0.000, C 0.000 }
gfCNCPoint3[9390] = {X 432.5144, Y 49.1600, Z -3.8333, A 0.000, B 0.000, C 0.000 }
gfCNCPoint3[9391] = {X 431.5887, Y 49.0557, Z -3.8333, A 0.000, B 0.000, C 0.000 }
gfCNCPoint3[9392] = {X 430.7095, Y 48.7480, Z -3.8333, A 0.000, B 0.000, C 0.000 }
gfCNCPoint3[9393] = {X 429.9207, Y 48.2524, Z -3.8333, A 0.000, B 0.000, C 0.000 }
gfCNCPoint3[9394] = {X 429.2620, Y 47.5937, Z -3.8333, A 0.000, B 0.000, C 0.000 }
gfCNCPoint3[9395] = {X 428.7664, Y 46.8050, Z -3.8333, A 0.000, B 0.000, C 0.000 }
gfCNCPoint3[9396] = {X 428.4587, Y 45.9257, Z -3.8333, A 0.000, B 0.000, C 0.000 }
gfCNCPoint3[9397] = {X 428.3544, Y 45.0000, Z -3.8333, A 0.000, B 0.000, C 0.000 }
gfCNCPoint3[9398] = {X 428.3548, Y 44.1516, Z -3.8333, A 0.000, B 0.000, C 0.000 }
gfCNCPoint3[9399] = {X 428.4510, Y 43.3174, Z -3.8333, A 0.000, B 0.000, C 0.000 }
gfCNCPoint3[9400] = {X 428.7128, Y 42.5195, Z -3.8333, A 0.000, B 0.000, C 0.000 }
gfCNCPoint3[9401] = {X 429.1295, Y 41.7905, Z -3.8333, A 0.000, B 0.000, C 0.000 }
gfCNCPoint3[9402] = {X 429.6841, Y 41.1600, Z -3.8333, A 0.000, B 0.000, C 0.000 }
gfCNCPoint3[9403] = {X 430.3541, Y 40.6537, Z -3.8333, A 0.000, B 0.000, C 0.000 }
gfCNCPoint3[9404] = {X 431.1120, Y 40.2923, Z -3.8333, A 0.000, B 0.000, C 0.000 }
gfCNCPoint3[9405] = {X 435.1989, Y 32.2927, Z -3.8333, A 0.000, B 0.000, C 0.000 }
gfCNCPoint3[9406] = {X 434.0150, Y 31.5179, Z -3.8333, A 0.000, B 0.000, C 0.000 }
gfCNCPoint3[9407] = {X 432.9386, Y 30.5996, Z -3.8333, A 0.000, B 0.000, C 0.000 }
gfCNCPoint3[9408] = {X 431.9870, Y 29.5524, Z -3.8333, A 0.000, B 0.000, C 0.000 }
gfCNCPoint3[9409] = {X 431.1756, Y 28.3933, Z -3.8333, A 0.000, B 0.000, C 0.000 }
gfCNCPoint3[9410] = {X 430.5173, Y 27.1408, Z -3.8333, A 0.000, B 0.000, C 0.000 }
gfCNCPoint3[9411] = {X 430.0227, Y 25.8152, Z -3.8333, A 0.000, B 0.000, C 0.000 }
gfCNCPoint3[9412] = {X 429.6079, Y 24.0214, Z -3.8333, A 0.000, B 0.000, C 0.000 }
gfCNCPoint3[9413] = {X 429.3965, Y 22.1925, Z -3.8333, A 0.000, B 0.000, C 0.000 }
gfCNCPoint3[9414] = {X 429.3913, Y 20.3513, Z -3.8333, A 0.000, B 0.000, C 0.000 }
gfCNCPoint3[9415] = {X 429.5923, Y 18.5212, Z -3.8333, A 0.000, B 0.000, C 0.000 }
gfCNCPoint3[9416] = {X 429.9969, Y 16.7251, Z -3.8333, A 0.000, B 0.000, C 0.000 }
gfCNCPoint3[9417] = {X 430.5114, Y 15.2752, Z -3.8333, A 0.000, B 0.000, C 0.000 }
gfCNCPoint3[9418] = {X 431.2126, Y 13.9058, Z -3.8333, A 0.000, B 0.000, C 0.000 }
gfCNCPoint3[9419] = {X 432.0884, Y 12.6409, Z -3.8333, A 0.000, B 0.000, C 0.000 }
gfCNCPoint3[9420] = {X 433.1235, Y 11.5026, Z -3.8333, A 0.000, B 0.000, C 0.000 }
gfCNCPoint3[9421] = {X 434.2996, Y 10.5109, Z -3.8333, A 0.000, B 0.000, C 0.000 }
gfCNCPoint3[9422] = {X 435.5964, Y 9.6830, Z -3.8333, A 0.000, B 0.000, C 0.000 }
gfCNCPoint3[9423] = {X 436.9910, Y 9.0334, Z -3.8333, A 0.000, B 0.000, C 0.000 }
gfCNCPoint3[9424] = {X 438.4592, Y 8.5736, Z -3.8333, A 0.000, B 0.000, C 0.000 }
gfCNCPoint3[9425] = {X 440.0719, Y 8.2675, Z -3.8333, A 0.000, B 0.000, C 0.000 }
gfCNCPoint3[9426] = {X 441.7036, Y 8.0876, Z -3.8333, A 0.000, B 0.000, C 0.000 }
gfCNCPoint3[9427] = {X 443.3443, Y 8.0350, Z -3.8333, A 0.000, B 0.000, C 0.000 }
gfCNCPoint3[9428] = {X 444.0362, Y 8.0309, Z -3.8333, A 0.000, B 0.000, C 0.000 }
gfCNCPoint3[9429] = {X 459.4467, Y 8.0309, Z -3.8333, A 0.000, B 0.000, C 0.000 }
gfCNCPoint3[9430] = {X 460.3704, Y 8.1350, Z -3.8333, A 0.000, B 0.000, C 0.000 }
gfCNCPoint3[9431] = {X 461.2478, Y 8.4420, Z -3.8333, A 0.000, B 0.000, C 0.000 }
gfCNCPoint3[9432] = {X 462.0349, Y 8.9366, Z -3.8333, A 0.000, B 0.000, C 0.000 }
gfCNCPoint3[9433] = {X 462.6923, Y 9.5939, Z -3.8333, A 0.000, B 0.000, C 0.000 }
gfCNCPoint3[9434] = {X 463.1868, Y 10.3810, Z -3.8333, A 0.000, B 0.000, C 0.000 }
gfCNCPoint3[9435] = {X 463.4939, Y 11.2584, Z -3.8333, A 0.000, B 0.000, C 0.000 }
gfCNCPoint3[9436] = {X 463.5979, Y 12.1822, Z -3.8333, A 0.000, B 0.000, C 0.000 }
gfCNCPoint3[9437] = {X 463.5979, Y 12.9781, Z -3.8333, A 0.000, B 0.000, C 0.000 }
gfCNCPoint3[9438] = {X 463.5022, Y 13.8652, Z -3.8333, A 0.000, B 0.000, C 0.000 }
gfCNCPoint3[9439] = {X 463.2196, Y 14.7114, Z -3.8333, A 0.000, B 0.000, C 0.000 }
gfCNCPoint3[9440] = {X 462.7630, Y 15.4779, Z -3.8333, A 0.000, B 0.000, C 0.000 }
gfCNCPoint3[9441] = {X 462.1535, Y 16.1294, Z -3.8333, A 0.000, B 0.000, C 0.000 }
gfCNCPoint3[9442] = {X 462.0703, Y 16.1992, Z -3.8333, A 0.000, B 0.000, C 0.000 }
gfCNCPoint3[9443] = {X 462.0705, Y 28.5935, Z -3.8333, A 0.000, B 0.000, C 0.000 }
gfCNCPoint3[9444] = {X 466.0705, Y 28.5935, Z -3.8333, A 0.000, B 0.000, C 0.000 }
gfCNCPoint3[9445] = {X 461.9905, Y 28.5935, Z -3.8333, A 0.000, B 0.000, C 0.000 }
gfCNCPoint3[9446] = {X 461.9908, Y 41.0274, Z -3.8333, A 0.000, B 0.000, C 0.000 }
gfCNCPoint3[9447] = {X 462.0858, Y 41.1047, Z -3.8333, A 0.000, B 0.000, C 0.000 }
gfCNCPoint3[9448] = {X 462.6846, Y 41.7378, Z -3.8333, A 0.000, B 0.000, C 0.000 }
gfCNCPoint3[9449] = {X 463.1353, Y 42.4837, Z -3.8333, A 0.000, B 0.000, C 0.000 }
gfCNCPoint3[9450] = {X 463.4173, Y 43.3082, Z -3.8333, A 0.000, B 0.000, C 0.000 }
gfCNCPoint3[9451] = {X 463.5178, Y 44.1738, Z -3.8333, A 0.000, B 0.000, C 0.000 }
gfCNCPoint3[9452] = {X 463.5179, Y 45.0000, Z -3.8333, A 0.000, B 0.000, C 0.000 }
gfCNCPoint3[9453] = {X 463.4156, Y 45.9079, Z -3.8333, A 0.000, B 0.000, C 0.000 }
gfCNCPoint3[9454] = {X 463.1139, Y 46.7702, Z -3.8333, A 0.000, B 0.000, C 0.000 }
gfCNCPoint3[9455] = {X 462.6278, Y 47.5438, Z -3.8333, A 0.000, B 0.000, C 0.000 }
gfCNCPoint3[9456] = {X 461.9818, Y 48.1899, Z -3.8333, A 0.000, B 0.000, C 0.000 }
gfCNCPoint3[9457] = {X 461.2082, Y 48.6760, Z -3.8333, A 0.000, B 0.000, C 0.000 }
gfCNCPoint3[9458] = {X 460.3458, Y 48.9777, Z -3.8333, A 0.000, B 0.000, C 0.000 }
gfCNCPoint3[9459] = {X 459.4379, Y 49.0800, Z -3.8333, A 0.000, B 0.000, C 0.000 }
gfCNCPoint3[9460] = {X 452.9945, Y 49.0800, Z -3.8333, A 0.000, B 0.000, C 0.000 }
gfCNCPoint3[9461] = {X 452.0912, Y 48.9788, Z -3.8333, A 0.000, B 0.000, C 0.000 }
gfCNCPoint3[9462] = {X 451.2327, Y 48.6800, Z -3.8333, A 0.000, B 0.000, C 0.000 }
gfCNCPoint3[9463] = {X 450.4617, Y 48.1987, Z -3.8333, A 0.000, B 0.000, C 0.000 }
gfCNCPoint3[9464] = {X 449.8164, Y 47.5585, Z -3.8333, A 0.000, B 0.000, C 0.000 }
gfCNCPoint3[9465] = {X 449.3288, Y 46.7914, Z -3.8333, A 0.000, B 0.000, C 0.000 }
gfCNCPoint3[9466] = {X 449.0232, Y 45.9354, Z -3.8333, A 0.000, B 0.000, C 0.000 }
gfCNCPoint3[9467] = {X 448.9146, Y 45.0330, Z -3.8333, A 0.000, B 0.000, C 0.000 }
gfCNCPoint3[9468] = {X 448.9149, Y 44.1527, Z -3.8333, A 0.000, B 0.000, C 0.000 }
gfCNCPoint3[9469] = {X 449.0254, Y 43.2637, Z -3.8333, A 0.000, B 0.000, C 0.000 }
gfCNCPoint3[9470] = {X 449.3274, Y 42.4203, Z -3.8333, A 0.000, B 0.000, C 0.000 }
gfCNCPoint3[9471] = {X 449.8061, Y 41.6631, Z -3.8333, A 0.000, B 0.000, C 0.000 }
gfCNCPoint3[9472] = {X 450.4384, Y 41.0287, Z -3.8333, A 0.000, B 0.000, C 0.000 }
gfCNCPoint3[9473] = {X 450.4384, Y 34.2338, Z -3.8333, A 0.000, B 0.000, C 0.000 }
gfCNCPoint3[9474] = {X 447.3278, Y 34.2338, Z -3.8333, A 0.000, B 0.000, C 0.000 }
gfCNCPoint3[9475] = {X 442.9279, Y 42.8004, Z -3.8333, A 0.000, B 0.000, C 0.000 }
gfCNCPoint3[9476] = {X 442.9681, Y 42.9097, Z -3.8333, A 0.000, B 0.000, C 0.000 }
gfCNCPoint3[9477] = {X 443.1241, Y 43.5327, Z -3.8333, A 0.000, B 0.000, C 0.000 }
gfCNCPoint3[9478] = {X 443.1803, Y 44.1725, Z -3.8333, A 0.000, B 0.000, C 0.000 }
gfCNCPoint3[9479] = {X 443.1805, Y 45.0000, Z -3.8333, A 0.000, B 0.000, C 0.000 }
gfCNCPoint3[9480] = {X 443.0782, Y 45.9079, Z -3.8333, A 0.000, B 0.000, C 0.000 }
gfCNCPoint3[9481] = {X 442.7764, Y 46.7702, Z -3.8333, A 0.000, B 0.000, C 0.000 }
gfCNCPoint3[9482] = {X 442.2903, Y 47.5438, Z -3.8333, A 0.000, B 0.000, C 0.000 }
gfCNCPoint3[9483] = {X 441.6443, Y 48.1899, Z -3.8333, A 0.000, B 0.000, C 0.000 }
gfCNCPoint3[9484] = {X 440.8707, Y 48.6760, Z -3.8333, A 0.000, B 0.000, C 0.000 }
gfCNCPoint3[9485] = {X 440.0084, Y 48.9777, Z -3.8333, A 0.000, B 0.000, C 0.000 }
gfCNCPoint3[9486] = {X 439.1005, Y 49.0800, Z -3.8333, A 0.000, B 0.000, C 0.000 }
gfCNCPoint3[9487] = {X 432.5144, Y 49.0800, Z -3.8333, A 0.000, B 0.000, C 0.000 }
gfCNCPoint3[9488] = {X 431.6065, Y 48.9777, Z -3.8333, A 0.000, B 0.000, C 0.000 }
gfCNCPoint3[9489] = {X 430.7442, Y 48.6760, Z -3.8333, A 0.000, B 0.000, C 0.000 }
gfCNCPoint3[9490] = {X 429.9706, Y 48.1899, Z -3.8333, A 0.000, B 0.000, C 0.000 }
gfCNCPoint3[9491] = {X 429.3245, Y 47.5438, Z -3.8333, A 0.000, B 0.000, C 0.000 }
gfCNCPoint3[9492] = {X 428.8385, Y 46.7702, Z -3.8333, A 0.000, B 0.000, C 0.000 }
gfCNCPoint3[9493] = {X 428.5367, Y 45.9079, Z -3.8333, A 0.000, B 0.000, C 0.000 }
gfCNCPoint3[9494] = {X 428.4344, Y 45.0000, Z -3.8333, A 0.000, B 0.000, C 0.000 }
gfCNCPoint3[9495] = {X 428.4348, Y 44.1527, Z -3.8333, A 0.000, B 0.000, C 0.000 }
gfCNCPoint3[9496] = {X 428.5303, Y 43.3294, Z -3.8333, A 0.000, B 0.000, C 0.000 }
gfCNCPoint3[9497] = {X 428.7902, Y 42.5424, Z -3.8333, A 0.000, B 0.000, C 0.000 }
gfCNCPoint3[9498] = {X 429.2038, Y 41.8242, Z -3.8333, A 0.000, B 0.000, C 0.000 }
gfCNCPoint3[9499] = {X 429.7540, Y 41.2044, Z -3.8333, A 0.000, B 0.000, C 0.000 }
gfCNCPoint3[9500] = {X 430.4181, Y 40.7085, Z -3.8333, A 0.000, B 0.000, C 0.000 }
gfCNCPoint3[9501] = {X 431.1687, Y 40.3571, Z -3.8333, A 0.000, B 0.000, C 0.000 }
gfCNCPoint3[9502] = {X 435.3051, Y 32.2607, Z -3.8333, A 0.000, B 0.000, C 0.000 }
gfCNCPoint3[9503] = {X 434.1141, Y 31.4920, Z -3.8333, A 0.000, B 0.000, C 0.000 }
gfCNCPoint3[9504] = {X 433.0310, Y 30.5776, Z -3.8333, A 0.000, B 0.000, C 0.000 }
gfCNCPoint3[9505] = {X 432.0735, Y 29.5323, Z -3.8333, A 0.000, B 0.000, C 0.000 }
gfCNCPoint3[9506] = {X 431.2572, Y 28.3734, Z -3.8333, A 0.000, B 0.000, C 0.000 }
gfCNCPoint3[9507] = {X 430.5955, Y 27.1198, Z -3.8333, A 0.000, B 0.000, C 0.000 }
gfCNCPoint3[9508] = {X 430.0993, Y 25.7920, Z -3.8333, A 0.000, B 0.000, C 0.000 }
gfCNCPoint3[9509] = {X 429.6866, Y 24.0071, Z -3.8333, A 0.000, B 0.000, C 0.000 }
gfCNCPoint3[9510] = {X 429.4764, Y 22.1872, Z -3.8333, A 0.000, B 0.000, C 0.000 }
gfCNCPoint3[9511] = {X 429.4712, Y 20.3552, Z -3.8333, A 0.000, B 0.000, C 0.000 }
gfCNCPoint3[9512] = {X 429.6712, Y 18.5342, Z -3.8333, A 0.000, B 0.000, C 0.000 }
gfCNCPoint3[9513] = {X 430.0739, Y 16.7470, Z -3.8333, A 0.000, B 0.000, C 0.000 }
gfCNCPoint3[9514] = {X 430.5848, Y 15.3070, Z -3.8333, A 0.000, B 0.000, C 0.000 }
gfCNCPoint3[9515] = {X 431.2812, Y 13.9470, Z -3.8333, A 0.000, B 0.000, C 0.000 }
gfCNCPoint3[9516] = {X 432.1510, Y 12.6908, Z -3.8333, A 0.000, B 0.000, C 0.000 }
gfCNCPoint3[9517] = {X 433.1789, Y 11.5603, Z -3.8333, A 0.000, B 0.000, C 0.000 }
gfCNCPoint3[9518] = {X 434.3470, Y 10.5754, Z -3.8333, A 0.000, B 0.000, C 0.000 }
gfCNCPoint3[9519] = {X 435.6348, Y 9.7531, Z -3.8333, A 0.000, B 0.000, C 0.000 }
gfCNCPoint3[9520] = {X 437.0199, Y 9.1080, Z -3.8333, A 0.000, B 0.000, C 0.000 }
gfCNCPoint3[9521] = {X 438.4780, Y 8.6513, Z -3.8333, A 0.000, B 0.000, C 0.000 }
gfCNCPoint3[9522] = {X 440.0845, Y 8.3465, Z -3.8333, A 0.000, B 0.000, C 0.000 }
gfCNCPoint3[9523] = {X 441.7099, Y 8.1673, Z -3.8333, A 0.000, B 0.000, C 0.000 }
gfCNCPoint3[9524] = {X 443.3442, Y 8.1150, Z -3.8333, A 0.000, B 0.000, C 0.000 }
gfCNCPoint3[9525] = {X 444.0364, Y 8.1109, Z -3.8333, A 0.000, B 0.000, C 0.000 }
gfCNCPoint3[9526] = {X 459.4467, Y 8.1109, Z -3.8333, A 0.000, B 0.000, C 0.000 }
gfCNCPoint3[9527] = {X 460.3526, Y 8.2130, Z -3.8333, A 0.000, B 0.000, C 0.000 }
gfCNCPoint3[9528] = {X 461.2131, Y 8.5141, Z -3.8333, A 0.000, B 0.000, C 0.000 }
gfCNCPoint3[9529] = {X 461.9851, Y 8.9991, Z -3.8333, A 0.000, B 0.000, C 0.000 }
gfCNCPoint3[9530] = {X 462.6297, Y 9.6438, Z -3.8333, A 0.000, B 0.000, C 0.000 }
gfCNCPoint3[9531] = {X 463.1148, Y 10.4157, Z -3.8333, A 0.000, B 0.000, C 0.000 }
gfCNCPoint3[9532] = {X 463.4159, Y 11.2762, Z -3.8333, A 0.000, B 0.000, C 0.000 }
gfCNCPoint3[9533] = {X 463.5179, Y 12.1822, Z -3.8333, A 0.000, B 0.000, C 0.000 }
gfCNCPoint3[9534] = {X 463.5179, Y 12.9781, Z -3.8333, A 0.000, B 0.000, C 0.000 }
gfCNCPoint3[9535] = {X 463.4241, Y 13.8481, Z -3.8333, A 0.000, B 0.000, C 0.000 }
gfCNCPoint3[9536] = {X 463.1469, Y 14.6781, Z -3.8333, A 0.000, B 0.000, C 0.000 }
gfCNCPoint3[9537] = {X 462.6991, Y 15.4298, Z -3.8333, A 0.000, B 0.000, C 0.000 }
gfCNCPoint3[9538] = {X 462.1013, Y 16.0688, Z -3.8333, A 0.000, B 0.000, C 0.000 }
gfCNCPoint3[9539] = {X 462.0439, Y 16.1174, Z -3.8333, A 0.000, B 0.000, C 0.000 }
gfCNCPoint3[9540] = {X 461.9856, Y 16.1649, Z -3.8333, A 0.000, B 0.000, C 0.000 }
gfCNCPoint3[9541] = {X 461.9903, Y 16.1992, Z -3.8333, A 0.000, B 0.000, C 0.000 }
gfCNCPoint3[9542] = {X 461.9905, Y 28.5935, Z -3.8333, A 0.000, B 0.000, C 0.000 }
gfCNCPoint3[9543] = {X 465.9905, Y 28.5935, Z -3.8333, A 0.000, B 0.000, C 0.000 }
gfCNCPoint3[9544] = {X 465.9905, Y 28.5934, Z -3.8333, A 0.000, B 0.000, C 0.000 }
gfCNCPoint3[9545] = {X 461.9102, Y 28.5935, Z -3.8333, A 0.000, B 0.000, C 0.000 }
gfCNCPoint3[9546] = {X 461.9108, Y 41.0655, Z -3.8333, A 0.000, B 0.000, C 0.000 }
gfCNCPoint3[9547] = {X 462.0496, Y 41.1790, Z -3.8333, A 0.000, B 0.000, C 0.000 }
gfCNCPoint3[9548] = {X 462.6355, Y 41.8055, Z -3.8333, A 0.000, B 0.000, C 0.000 }
gfCNCPoint3[9549] = {X 463.0743, Y 42.5425, Z -3.8333, A 0.000, B 0.000, C 0.000 }
gfCNCPoint3[9550] = {X 463.3460, Y 43.3561, Z -3.8333, A 0.000, B 0.000, C 0.000 }
gfCNCPoint3[9551] = {X 463.4379, Y 44.2089, Z -3.8333, A 0.000, B 0.000, C 0.000 }
gfCNCPoint3[9552] = {X 463.4379, Y 45.0000, Z -3.8333, A 0.000, B 0.000, C 0.000 }
gfCNCPoint3[9553] = {X 463.3377, Y 45.8901, Z -3.8333, A 0.000, B 0.000, C 0.000 }
gfCNCPoint3[9554] = {X 463.0418, Y 46.7355, Z -3.8333, A 0.000, B 0.000, C 0.000 }
gfCNCPoint3[9555] = {X 462.5653, Y 47.4940, Z -3.8333, A 0.000, B 0.000, C 0.000 }
gfCNCPoint3[9556] = {X 461.9319, Y 48.1273, Z -3.8333, A 0.000, B 0.000, C 0.000 }
gfCNCPoint3[9557] = {X 461.1735, Y 48.6039, Z -3.8333, A 0.000, B 0.000, C 0.000 }
gfCNCPoint3[9558] = {X 460.3280, Y 48.8997, Z -3.8333, A 0.000, B 0.000, C 0.000 }
gfCNCPoint3[9559] = {X 459.4379, Y 49.0000, Z -3.8333, A 0.000, B 0.000, C 0.000 }
gfCNCPoint3[9560] = {X 452.9945, Y 49.0000, Z -3.8333, A 0.000, B 0.000, C 0.000 }
gfCNCPoint3[9561] = {X 452.1044, Y 48.8997, Z -3.8333, A 0.000, B 0.000, C 0.000 }
gfCNCPoint3[9562] = {X 451.2589, Y 48.6039, Z -3.8333, A 0.000, B 0.000, C 0.000 }
gfCNCPoint3[9563] = {X 450.5005, Y 48.1273, Z -3.8333, A 0.000, B 0.000, C 0.000 }
gfCNCPoint3[9564] = {X 449.8671, Y 47.4939, Z -3.8333, A 0.000, B 0.000, C 0.000 }
gfCNCPoint3[9565] = {X 449.3906, Y 46.7355, Z -3.8333, A 0.000, B 0.000, C 0.000 }
gfCNCPoint3[9566] = {X 449.0948, Y 45.8900, Z -3.8333, A 0.000, B 0.000, C 0.000 }
gfCNCPoint3[9567] = {X 448.9945, Y 45.0000, Z -3.8333, A 0.000, B 0.000, C 0.000 }
gfCNCPoint3[9568] = {X 448.9949, Y 44.1538, Z -3.8333, A 0.000, B 0.000, C 0.000 }
gfCNCPoint3[9569] = {X 449.1055, Y 43.2730, Z -3.8333, A 0.000, B 0.000, C 0.000 }
gfCNCPoint3[9570] = {X 449.4077, Y 42.4382, Z -3.8333, A 0.000, B 0.000, C 0.000 }
gfCNCPoint3[9571] = {X 449.8865, Y 41.6907, Z -3.8333, A 0.000, B 0.000, C 0.000 }
gfCNCPoint3[9572] = {X 450.5184, Y 41.0672, Z -3.8333, A 0.000, B 0.000, C 0.000 }
gfCNCPoint3[9573] = {X 450.5184, Y 34.1538, Z -3.8333, A 0.000, B 0.000, C 0.000 }
gfCNCPoint3[9574] = {X 447.5232, Y 34.1538, Z -3.8333, A 0.000, B 0.000, C 0.000 }
gfCNCPoint3[9575] = {X 447.2794, Y 34.1529, Z -3.8333, A 0.000, B 0.000, C 0.000 }
gfCNCPoint3[9576] = {X 442.8407, Y 42.7951, Z -3.8333, A 0.000, B 0.000, C 0.000 }
gfCNCPoint3[9577] = {X 442.8967, Y 42.9484, Z -3.8333, A 0.000, B 0.000, C 0.000 }
gfCNCPoint3[9578] = {X 443.0492, Y 43.5705, Z -3.8333, A 0.000, B 0.000, C 0.000 }
gfCNCPoint3[9579] = {X 443.1005, Y 44.2089, Z -3.8333, A 0.000, B 0.000, C 0.000 }
gfCNCPoint3[9580] = {X 443.1005, Y 45.0000, Z -3.8333, A 0.000, B 0.000, C 0.000 }
gfCNCPoint3[9581] = {X 443.0002, Y 45.8901, Z -3.8333, A 0.000, B 0.000, C 0.000 }
gfCNCPoint3[9582] = {X 442.7043, Y 46.7355, Z -3.8333, A 0.000, B 0.000, C 0.000 }
gfCNCPoint3[9583] = {X 442.2278, Y 47.4940, Z -3.8333, A 0.000, B 0.000, C 0.000 }
gfCNCPoint3[9584] = {X 441.5944, Y 48.1273, Z -3.8333, A 0.000, B 0.000, C 0.000 }
gfCNCPoint3[9585] = {X 440.8360, Y 48.6039, Z -3.8333, A 0.000, B 0.000, C 0.000 }
gfCNCPoint3[9586] = {X 439.9906, Y 48.8997, Z -3.8333, A 0.000, B 0.000, C 0.000 }
gfCNCPoint3[9587] = {X 439.1005, Y 49.0000, Z -3.8333, A 0.000, B 0.000, C 0.000 }
gfCNCPoint3[9588] = {X 432.5144, Y 49.0000, Z -3.8333, A 0.000, B 0.000, C 0.000 }
gfCNCPoint3[9589] = {X 431.6243, Y 48.8997, Z -3.8333, A 0.000, B 0.000, C 0.000 }
gfCNCPoint3[9590] = {X 430.7789, Y 48.6039, Z -3.8333, A 0.000, B 0.000, C 0.000 }
gfCNCPoint3[9591] = {X 430.0204, Y 48.1273, Z -3.8333, A 0.000, B 0.000, C 0.000 }
gfCNCPoint3[9592] = {X 429.3871, Y 47.4940, Z -3.8333, A 0.000, B 0.000, C 0.000 }
gfCNCPoint3[9593] = {X 428.9105, Y 46.7355, Z -3.8333, A 0.000, B 0.000, C 0.000 }
gfCNCPoint3[9594] = {X 428.6147, Y 45.8901, Z -3.8333, A 0.000, B 0.000, C 0.000 }
gfCNCPoint3[9595] = {X 428.5144, Y 45.0000, Z -3.8333, A 0.000, B 0.000, C 0.000 }
gfCNCPoint3[9596] = {X 428.5148, Y 44.1538, Z -3.8333, A 0.000, B 0.000, C 0.000 }
gfCNCPoint3[9597] = {X 428.6096, Y 43.3414, Z -3.8333, A 0.000, B 0.000, C 0.000 }
gfCNCPoint3[9598] = {X 428.8676, Y 42.5654, Z -3.8333, A 0.000, B 0.000, C 0.000 }
gfCNCPoint3[9599] = {X 429.2781, Y 41.8580, Z -3.8333, A 0.000, B 0.000, C 0.000 }
gfCNCPoint3[9600] = {X 429.8239, Y 41.2489, Z -3.8333, A 0.000, B 0.000, C 0.000 }
gfCNCPoint3[9601] = {X 430.4821, Y 40.7635, Z -3.8333, A 0.000, B 0.000, C 0.000 }
gfCNCPoint3[9602] = {X 431.2253, Y 40.4222, Z -3.8333, A 0.000, B 0.000, C 0.000 }
gfCNCPoint3[9603] = {X 435.4115, Y 32.2282, Z -3.8333, A 0.000, B 0.000, C 0.000 }
gfCNCPoint3[9604] = {X 434.2134, Y 31.4658, Z -3.8333, A 0.000, B 0.000, C 0.000 }
gfCNCPoint3[9605] = {X 433.1236, Y 30.5554, Z -3.8333, A 0.000, B 0.000, C 0.000 }
gfCNCPoint3[9606] = {X 432.1600, Y 29.5122, Z -3.8333, A 0.000, B 0.000, C 0.000 }
gfCNCPoint3[9607] = {X 431.3389, Y 28.3536, Z -3.8333, A 0.000, B 0.000, C 0.000 }
gfCNCPoint3[9608] = {X 430.6738, Y 27.0988, Z -3.8333, A 0.000, B 0.000, C 0.000 }
gfCNCPoint3[9609] = {X 430.1759, Y 25.7689, Z -3.8333, A 0.000, B 0.000, C 0.000 }
gfCNCPoint3[9610] = {X 429.7653, Y 23.9928, Z -3.8333, A 0.000, B 0.000, C 0.000 }
gfCNCPoint3[9611] = {X 429.5562, Y 22.1819, Z -3.8333, A 0.000, B 0.000, C 0.000 }
gfCNCPoint3[9612] = {X 429.5511, Y 20.3591, Z -3.8333, A 0.000, B 0.000, C 0.000 }
gfCNCPoint3[9613] = {X 429.7502, Y 18.5471, Z -3.8333, A 0.000, B 0.000, C 0.000 }
gfCNCPoint3[9614] = {X 430.1509, Y 16.7687, Z -3.8333, A 0.000, B 0.000, C 0.000 }
gfCNCPoint3[9615] = {X 430.6582, Y 15.3387, Z -3.8333, A 0.000, B 0.000, C 0.000 }
gfCNCPoint3[9616] = {X 431.3498, Y 13.9881, Z -3.8333, A 0.000, B 0.000, C 0.000 }
gfCNCPoint3[9617] = {X 432.2136, Y 12.7406, Z -3.8333, A 0.000, B 0.000, C 0.000 }
gfCNCPoint3[9618] = {X 433.2344, Y 11.6180, Z -3.8333, A 0.000, B 0.000, C 0.000 }
gfCNCPoint3[9619] = {X 434.3944, Y 10.6398, Z -3.8333, A 0.000, B 0.000, C 0.000 }
gfCNCPoint3[9620] = {X 435.6733, Y 9.8233, Z -3.8333, A 0.000, B 0.000, C 0.000 }
gfCNCPoint3[9621] = {X 437.0488, Y 9.1826, Z -3.8333, A 0.000, B 0.000, C 0.000 }
gfCNCPoint3[9622] = {X 438.4968, Y 8.7291, Z -3.8333, A 0.000, B 0.000, C 0.000 }
gfCNCPoint3[9623] = {X 440.0971, Y 8.4255, Z -3.8333, A 0.000, B 0.000, C 0.000 }
gfCNCPoint3[9624] = {X 441.7162, Y 8.2471, Z -3.8333, A 0.000, B 0.000, C 0.000 }
gfCNCPoint3[9625] = {X 443.3442, Y 8.1950, Z -3.8333, A 0.000, B 0.000, C 0.000 }
gfCNCPoint3[9626] = {X 444.0367, Y 8.1909, Z -3.8333, A 0.000, B 0.000, C 0.000 }
gfCNCPoint3[9627] = {X 459.4467, Y 8.1909, Z -3.8333, A 0.000, B 0.000, C 0.000 }
gfCNCPoint3[9628] = {X 460.3348, Y 8.2910, Z -3.8333, A 0.000, B 0.000, C 0.000 }
gfCNCPoint3[9629] = {X 461.1784, Y 8.5862, Z -3.8333, A 0.000, B 0.000, C 0.000 }
gfCNCPoint3[9630] = {X 461.9352, Y 9.0617, Z -3.8333, A 0.000, B 0.000, C 0.000 }
gfCNCPoint3[9631] = {X 462.5672, Y 9.6937, Z -3.8333, A 0.000, B 0.000, C 0.000 }
gfCNCPoint3[9632] = {X 463.0427, Y 10.4504, Z -3.8333, A 0.000, B 0.000, C 0.000 }
gfCNCPoint3[9633] = {X 463.3379, Y 11.2940, Z -3.8333, A 0.000, B 0.000, C 0.000 }
gfCNCPoint3[9634] = {X 463.4379, Y 12.1822, Z -3.8333, A 0.000, B 0.000, C 0.000 }
gfCNCPoint3[9635] = {X 463.4378, Y 13.0163, Z -3.8333, A 0.000, B 0.000, C 0.000 }
gfCNCPoint3[9636] = {X 463.3397, Y 13.8590, Z -3.8333, A 0.000, B 0.000, C 0.000 }
gfCNCPoint3[9637] = {X 463.0662, Y 14.6621, Z -3.8333, A 0.000, B 0.000, C 0.000 }
gfCNCPoint3[9638] = {X 462.6294, Y 15.3894, Z -3.8333, A 0.000, B 0.000, C 0.000 }
gfCNCPoint3[9639] = {X 462.0491, Y 16.0082, Z -3.8333, A 0.000, B 0.000, C 0.000 }
gfCNCPoint3[9640] = {X 461.9724, Y 16.0726, Z -3.8333, A 0.000, B 0.000, C 0.000 }
gfCNCPoint3[9641] = {X 461.8942, Y 16.1351, Z -3.8333, A 0.000, B 0.000, C 0.000 }
gfCNCPoint3[9642] = {X 461.9103, Y 16.1928, Z -3.8333, A 0.000, B 0.000, C 0.000 }
gfCNCPoint3[9643] = {X 461.9096, Y 16.7687, Z -3.8333, A 0.000, B 0.000, C 0.000 }
gfCNCPoint3[9644] = {X 461.9102, Y 28.5935, Z -3.8333, A 0.000, B 0.000, C 0.000 }
gfCNCPoint3[9645] = {X 465.9905, Y 28.5934, Z -3.8333, A 0.000, B 0.000, C 0.000 }
gfCNCPoint3[9646] = {X 465.9905, Y 28.5934, Z -0.8333, A 0.000, B 0.000, C 0.000 }
gfCNCPoint3[9647] = {X 465.9905, Y 28.5934, Z 11.0000, A 0.000, B 0.000, C 0.000 }
gfCNCPoint3[9648] = {X 492.3835, Y 3.7909, Z 11.0000, A 0.000, B 0.000, C 0.000 }
gfCNCPoint3[9649] = {X 492.3835, Y 3.7909, Z -0.8333, A 0.000, B 0.000, C 0.000 }
gfCNCPoint3[9650] = {X 492.3835, Y 3.7909, Z -3.8333, A 0.000, B 0.000, C 0.000 }
gfCNCPoint3[9651] = {X 492.3835, Y 7.8709, Z -3.8333, A 0.000, B 0.000, C 0.000 }
gfCNCPoint3[9652] = {X 502.2066, Y 7.8709, Z -3.8333, A 0.000, B 0.000, C 0.000 }
gfCNCPoint3[9653] = {X 502.7394, Y 7.8751, Z -3.8333, A 0.000, B 0.000, C 0.000 }
gfCNCPoint3[9654] = {X 503.6913, Y 7.9893, Z -3.8333, A 0.000, B 0.000, C 0.000 }
gfCNCPoint3[9655] = {X 504.5943, Y 8.3115, Z -3.8333, A 0.000, B 0.000, C 0.000 }
gfCNCPoint3[9656] = {X 505.4035, Y 8.8257, Z -3.8333, A 0.000, B 0.000, C 0.000 }
gfCNCPoint3[9657] = {X 506.0787, Y 9.5062, Z -3.8333, A 0.000, B 0.000, C 0.000 }
gfCNCPoint3[9658] = {X 506.5865, Y 10.3194, Z -3.8333, A 0.000, B 0.000, C 0.000 }
gfCNCPoint3[9659] = {X 506.9017, Y 11.2249, Z -3.8333, A 0.000, B 0.000, C 0.000 }
gfCNCPoint3[9660] = {X 507.0085, Y 12.1776, Z -3.8333, A 0.000, B 0.000, C 0.000 }
gfCNCPoint3[9661] = {X 507.0085, Y 12.9781, Z -3.8333, A 0.000, B 0.000, C 0.000 }
gfCNCPoint3[9662] = {X 506.9072, Y 13.9082, Z -3.8333, A 0.000, B 0.000, C 0.000 }
gfCNCPoint3[9663] = {X 506.6080, Y 14.7946, Z -3.8333, A 0.000, B 0.000, C 0.000 }
gfCNCPoint3[9664] = {X 506.1250, Y 15.5958, Z -3.8333, A 0.000, B 0.000, C 0.000 }
gfCNCPoint3[9665] = {X 505.4809, Y 16.2742, Z -3.8333, A 0.000, B 0.000, C 0.000 }
gfCNCPoint3[9666] = {X 505.4808, Y 40.9125, Z -3.8333, A 0.000, B 0.000, C 0.000 }
gfCNCPoint3[9667] = {X 506.1193, Y 41.5836, Z -3.8333, A 0.000, B 0.000, C 0.000 }
gfCNCPoint3[9668] = {X 506.6001, Y 42.3753, Z -3.8333, A 0.000, B 0.000, C 0.000 }
gfCNCPoint3[9669] = {X 506.9010, Y 43.2513, Z -3.8333, A 0.000, B 0.000, C 0.000 }
gfCNCPoint3[9670] = {X 507.0083, Y 44.1713, Z -3.8333, A 0.000, B 0.000, C 0.000 }
gfCNCPoint3[9671] = {X 507.0085, Y 45.0000, Z -3.8333, A 0.000, B 0.000, C 0.000 }
gfCNCPoint3[9672] = {X 506.9002, Y 45.9613, Z -3.8333, A 0.000, B 0.000, C 0.000 }
gfCNCPoint3[9673] = {X 506.5807, Y 46.8744, Z -3.8333, A 0.000, B 0.000, C 0.000 }
gfCNCPoint3[9674] = {X 506.0660, Y 47.6935, Z -3.8333, A 0.000, B 0.000, C 0.000 }
gfCNCPoint3[9675] = {X 505.3820, Y 48.3775, Z -3.8333, A 0.000, B 0.000, C 0.000 }
gfCNCPoint3[9676] = {X 504.5629, Y 48.8922, Z -3.8333, A 0.000, B 0.000, C 0.000 }
gfCNCPoint3[9677] = {X 503.6498, Y 49.2117, Z -3.8333, A 0.000, B 0.000, C 0.000 }
